// waga 
eWeightPackage2PhasePackageState[2].nID; eWeightPackage2PhasePackageState[2].nCardNumber; eWeightPackage2PhasePackageState[2].bFormPresent; eWeightPackage2PhasePackageState[2].bBottlePresent; eWeightPackage2PhasePackageState[2].bWeightOK; eWeightPackage2PhasePackageState[2].bWeighed;	eWeightPackage2PhasePackageState[2].bDosingTwoPhases; eWeightPackage2PhasePackageState[2].lrDoseVolumeSV; eWeightPackage2PhasePackageState[2].lrDoseVolumeSVSecondPhase;  eWeightPackage2PhasePackageState[2].lrDoseVolumeCV; eWeightPackage2PhasePackageState[2].lrDoseVolumeCVSecondPhase; eWeightPackage2PhasePackageState[2].nDispencerNr; eWeightPackage2PhasePackageState[2].nDispencerNrSecondPhase; eWeightPackage2PhasePackageState[2].tDispencingTime; eWeightPackage2PhasePackageState[2].tDispencingTimeSecondPhase; eWeightPackage2PhasePackageState[2].bWeighed; eWeightPackage2PhasePackageState[2].bWeightOK; eWeightPackage2PhasePackageState[2].lrWeightSV; eWeightPackage2PhasePackageState[2].lrWeightMeasuredCV; eWeightPackage2PhasePackageState[2].lrWeightCV;
eWeightPackage2PhasePackageState[1].nID; eWeightPackage2PhasePackageState[1].nCardNumber; eWeightPackage2PhasePackageState[1].bFormPresent; eWeightPackage2PhasePackageState[1].bBottlePresent; eWeightPackage2PhasePackageState[1].bWeightOK; eWeightPackage2PhasePackageState[1].bWeighed;;	eWeightPackage2PhasePackageState[1].bDosingTwoPhases; eWeightPackage2PhasePackageState[1].lrDoseVolumeSV; eWeightPackage2PhasePackageState[1].lrDoseVolumeSVSecondPhase;  eWeightPackage2PhasePackageState[1].lrDoseVolumeCV; eWeightPackage2PhasePackageState[1].lrDoseVolumeCVSecondPhase; eWeightPackage2PhasePackageState[1].nDispencerNr; eWeightPackage2PhasePackageState[1].nDispencerNrSecondPhase; eWeightPackage2PhasePackageState[1].tDispencingTime; eWeightPackage2PhasePackageState[1].tDispencingTimeSecondPhase; eWeightPackage2PhasePackageState[1].bWeighed; eWeightPackage2PhasePackageState[1].bWeightOK; eWeightPackage2PhasePackageState[1].lrWeightSV; eWeightPackage2PhasePackageState[1].lrWeightMeasuredCV; eWeightPackage2PhasePackageState[1].lrWeightCV;


/////////////////////////////////////////////////

//[1..4] Strukutra pod wagą 
eWeightPackageState[4].nID; eWeightPackageState[4].nCardNumber; eWeightPackageState[4].bFormPresent; eWeightPackageState[4].bBottlePresent; eWeightPackageState[4].bWeightOK; eWeightPackageState[4].bWeighed; 	eWeightPackageState[4].bDosingTwoPhases; eWeightPackageState[4].lrDoseVolumeSV; eWeightPackageState[4].lrDoseVolumeSVSecondPhase;  eWeightPackageState[4].lrDoseVolumeCV; eWeightPackageState[4].lrDoseVolumeCVSecondPhase; eWeightPackageState[4].nDispencerNr; eWeightPackageState[4].nDispencerNrSecondPhase; eWeightPackageState[4].tDispencingTime; eWeightPackageState[4].tDispencingTimeSecondPhase; eWeightPackageState[4].bWeighed; eWeightPackageState[4].bWeightOK; eWeightPackageState[4].lrWeightSV; eWeightPackageState[4].lrWeightMeasuredCV; eWeightPackageState[4].lrWeightCV;
eWeightPackageState[3].nID; eWeightPackageState[3].nCardNumber; eWeightPackageState[3].bFormPresent; eWeightPackageState[3].bBottlePresent; eWeightPackageState[3].bWeightOK; eWeightPackageState[3].bWeighed; 	eWeightPackageState[3].bDosingTwoPhases; eWeightPackageState[3].lrDoseVolumeSV; eWeightPackageState[3].lrDoseVolumeSVSecondPhase;  eWeightPackageState[3].lrDoseVolumeCV; eWeightPackageState[3].lrDoseVolumeCVSecondPhase; eWeightPackageState[3].nDispencerNr; eWeightPackageState[3].nDispencerNrSecondPhase; eWeightPackageState[3].tDispencingTime; eWeightPackageState[3].tDispencingTimeSecondPhase; eWeightPackageState[3].bWeighed; eWeightPackageState[3].bWeightOK; eWeightPackageState[3].lrWeightSV; eWeightPackageState[3].lrWeightMeasuredCV; eWeightPackageState[3].lrWeightCV;
eWeightPackageState[2].nID; eWeightPackageState[2].nCardNumber; eWeightPackageState[2].bFormPresent; eWeightPackageState[2].bBottlePresent; eWeightPackageState[2].bWeightOK; eWeightPackageState[2].bWeighed;	eWeightPackageState[2].bDosingTwoPhases; eWeightPackageState[2].lrDoseVolumeSV; eWeightPackageState[2].lrDoseVolumeSVSecondPhase;  eWeightPackageState[2].lrDoseVolumeCV; eWeightPackageState[2].lrDoseVolumeCVSecondPhase; eWeightPackageState[2].nDispencerNr; eWeightPackageState[2].nDispencerNrSecondPhase; eWeightPackageState[2].tDispencingTime; eWeightPackageState[2].tDispencingTimeSecondPhase; eWeightPackageState[2].bWeighed; eWeightPackageState[2].bWeightOK; eWeightPackageState[2].lrWeightSV; eWeightPackageState[2].lrWeightMeasuredCV; eWeightPackageState[2].lrWeightCV;
eWeightPackageState[1].nID; eWeightPackageState[1].nCardNumber; eWeightPackageState[1].bFormPresent; eWeightPackageState[1].bBottlePresent; eWeightPackageState[1].bWeightOK; eWeightPackageState[1].bWeighed;;	eWeightPackageState[1].bDosingTwoPhases; eWeightPackageState[1].lrDoseVolumeSV; eWeightPackageState[1].lrDoseVolumeSVSecondPhase;  eWeightPackageState[1].lrDoseVolumeCV; eWeightPackageState[1].lrDoseVolumeCVSecondPhase; eWeightPackageState[1].nDispencerNr; eWeightPackageState[1].nDispencerNrSecondPhase; eWeightPackageState[1].tDispencingTime; eWeightPackageState[1].tDispencingTimeSecondPhase; eWeightPackageState[1].bWeighed; eWeightPackageState[1].bWeightOK; eWeightPackageState[1].lrWeightSV; eWeightPackageState[1].lrWeightMeasuredCV; eWeightPackageState[1].lrWeightCV;
															
eTempState1[1].nID; eTempState1[1].nCardNumber; eTempState1[1].bFormPresent;

eBeforeLidFeeder2PackageState[4].nID;eBeforeLidFeeder2PackageState[4].nCardNumber;eBeforeLidFeeder2PackageState[4].bFormPresent;eBeforeLidFeeder2PackageState[4].bBottlePresent;eBeforeLidFeeder2PackageState[4].bLidPutted;eBeforeLidFeeder2PackageState[4].bLidPutAborted;eBeforeLidFeeder2PackageState[4].bLidPuttedOK;eBeforeLidFeeder2PackageState[4].bLidPuttedChecked;eBeforeLidFeeder2PackageState[4].bLidSealed;eBeforeLidFeeder2PackageState[4].bLidSealingAborted;
eBeforeLidFeeder2PackageState[3].nID;eBeforeLidFeeder2PackageState[3].nCardNumber;eBeforeLidFeeder2PackageState[3].bFormPresent;eBeforeLidFeeder2PackageState[3].bBottlePresent;eBeforeLidFeeder2PackageState[3].bLidPutted;eBeforeLidFeeder2PackageState[3].bLidPutAborted;eBeforeLidFeeder2PackageState[3].bLidPuttedOK;eBeforeLidFeeder2PackageState[3].bLidPuttedChecked;eBeforeLidFeeder2PackageState[3].bLidSealed;eBeforeLidFeeder2PackageState[3].bLidSealingAborted;
eBeforeLidFeeder2PackageState[2].nID;eBeforeLidFeeder2PackageState[2].nCardNumber;eBeforeLidFeeder2PackageState[2].bFormPresent;eBeforeLidFeeder2PackageState[2].bBottlePresent;eBeforeLidFeeder2PackageState[2].bLidPutted;eBeforeLidFeeder2PackageState[2].bLidPutAborted;eBeforeLidFeeder2PackageState[2].bLidPuttedOK;eBeforeLidFeeder2PackageState[2].bLidPuttedChecked;eBeforeLidFeeder2PackageState[2].bLidSealed;eBeforeLidFeeder2PackageState[2].bLidSealingAborted;
eBeforeLidFeeder2PackageState[1].nID;eBeforeLidFeeder2PackageState[1].nCardNumber;eBeforeLidFeeder2PackageState[1].bFormPresent;eBeforeLidFeeder2PackageState[1].bBottlePresent;eBeforeLidFeeder2PackageState[1].bLidPutted;eBeforeLidFeeder2PackageState[1].bLidPutAborted;eBeforeLidFeeder2PackageState[1].bLidPuttedOK;eBeforeLidFeeder2PackageState[1].bLidPuttedChecked;eBeforeLidFeeder2PackageState[1].bLidSealed;eBeforeLidFeeder2PackageState[1].bLidSealingAborted;

eBeforeLidFeederPackageState[2].nID;eBeforeLidFeederPackageState[2].nCardNumber;eBeforeLidFeederPackageState[2].bFormPresent;eBeforeLidFeederPackageState[2].bBottlePresent;eBeforeLidFeederPackageState[2].bLidPutted;eBeforeLidFeederPackageState[2].bLidPutAborted;eBeforeLidFeederPackageState[2].bLidPuttedOK;eBeforeLidFeederPackageState[2].bLidPuttedChecked;eBeforeLidFeederPackageState[2].bLidSealed;eBeforeLidFeederPackageState[2].bLidSealingAborted;
eBeforeLidFeederPackageState[1].nID;eBeforeLidFeederPackageState[1].nCardNumber;eBeforeLidFeederPackageState[1].bFormPresent;eBeforeLidFeederPackageState[1].bBottlePresent;eBeforeLidFeederPackageState[1].bLidPutted;eBeforeLidFeederPackageState[1].bLidPutAborted;eBeforeLidFeederPackageState[1].bLidPuttedOK;eBeforeLidFeederPackageState[1].bLidPuttedChecked;eBeforeLidFeederPackageState[1].bLidSealed;eBeforeLidFeederPackageState[1].bLidSealingAborted;

eLidFeederPackageState[2].nID;eLidFeederPackageState[2].nCardNumber;eLidFeederPackageState[2].bFormPresent;eLidFeederPackageState[2].bBottlePresent;eLidFeederPackageState[2].bLidPutted;eLidFeederPackageState[2].bLidPutAborted;eLidFeederPackageState[2].bLidPuttedOK;eLidFeederPackageState[2].bLidPuttedChecked;eLidFeederPackageState[2].bLidSealed;eLidFeederPackageState[2].bLidSealingAborted;
eLidFeederPackageState[1].nID;eLidFeederPackageState[1].nCardNumber;eLidFeederPackageState[1].bFormPresent;eLidFeederPackageState[1].bBottlePresent;eLidFeederPackageState[1].bLidPutted;eLidFeederPackageState[1].bLidPutAborted;eLidFeederPackageState[1].bLidPuttedOK;eLidFeederPackageState[1].bLidPuttedChecked;eLidFeederPackageState[1].bLidSealed;eLidFeederPackageState[1].bLidSealingAborted;

eAfterLidFeederPackageState[2].nID;eAfterLidFeederPackageState[2].nCardNumber;eAfterLidFeederPackageState[2].bFormPresent;eAfterLidFeederPackageState[2].bBottlePresent;eAfterLidFeederPackageState[2].bLidPutted;eAfterLidFeederPackageState[2].bLidPutAborted;eAfterLidFeederPackageState[2].bLidPuttedOK;eAfterLidFeederPackageState[2].bLidPuttedChecked;eAfterLidFeederPackageState[2].bLidSealed;eAfterLidFeederPackageState[2].bLidSealingAborted;
eAfterLidFeederPackageState[1].nID;eAfterLidFeederPackageState[1].nCardNumber;eAfterLidFeederPackageState[1].bFormPresent;eAfterLidFeederPackageState[1].bBottlePresent;eAfterLidFeederPackageState[1].bLidPutted;eAfterLidFeederPackageState[1].bLidPutAborted;eAfterLidFeederPackageState[1].bLidPuttedOK;eAfterLidFeederPackageState[1].bLidPuttedChecked;eAfterLidFeederPackageState[1].bLidSealed;eAfterLidFeederPackageState[1].bLidSealingAborted;

eBeforeLidSealerPackageState[2].nID;eBeforeLidSealerPackageState[2].nCardNumber;eBeforeLidSealerPackageState[2].bFormPresent;eBeforeLidSealerPackageState[2].bBottlePresent;eBeforeLidSealerPackageState[2].bLidPutted;eBeforeLidSealerPackageState[2].bLidPutAborted;eBeforeLidSealerPackageState[2].bLidPuttedOK;eBeforeLidSealerPackageState[2].bLidPuttedChecked;eBeforeLidSealerPackageState[2].bLidSealed;eBeforeLidSealerPackageState[2].bLidSealingAborted;
eBeforeLidSealerPackageState[1].nID;eBeforeLidSealerPackageState[1].nCardNumber;eBeforeLidSealerPackageState[1].bFormPresent;eBeforeLidSealerPackageState[1].bBottlePresent;eBeforeLidSealerPackageState[1].bLidPutted;eBeforeLidSealerPackageState[1].bLidPutAborted;eBeforeLidSealerPackageState[1].bLidPuttedOK;eBeforeLidSealerPackageState[1].bLidPuttedChecked;eBeforeLidSealerPackageState[1].bLidSealed;eBeforeLidSealerPackageState[1].bLidSealingAborted;

eLidSealerPackageState[2].nID;eLidSealerPackageState[2].nCardNumber;eLidSealerPackageState[2].bFormPresent;eLidSealerPackageState[2].bBottlePresent;eLidSealerPackageState[2].bLidPutted;eLidSealerPackageState[2].bLidPutAborted;eLidSealerPackageState[2].bLidPuttedOK;eLidSealerPackageState[2].bLidPuttedChecked;eLidSealerPackageState[2].bLidSealed;eLidSealerPackageState[2].bLidSealingAborted;
eLidSealerPackageState[1].nID;eLidSealerPackageState[1].nCardNumber;eLidSealerPackageState[1].bFormPresent;eLidSealerPackageState[1].bBottlePresent;eLidSealerPackageState[1].bLidPutted;eLidSealerPackageState[1].bLidPutAborted;eLidSealerPackageState[1].bLidPuttedOK;eLidSealerPackageState[1].bLidPuttedChecked;eLidSealerPackageState[1].bLidSealed;eLidSealerPackageState[1].bLidSealingAborted;



eBeforeGateCapSorterPackageState[1].nID;	eBeforeGateCapSorterPackageState[1].nCardNumber;	eBeforeGateCapSorterPackageState[1].bFormPresent;

eBeforeCapSorterPackageState[4].nID;	eBeforeCapSorterPackageState[4].nCardNumber;	eBeforeCapSorterPackageState[4].bFormPresent;eBeforeCapSorterPackageState[4].bBottlePresent;
eBeforeCapSorterPackageState[3].nID;	eBeforeCapSorterPackageState[3].nCardNumber;	eBeforeCapSorterPackageState[3].bFormPresent;eBeforeCapSorterPackageState[3].bBottlePresent;
eBeforeCapSorterPackageState[2].nID;	eBeforeCapSorterPackageState[2].nCardNumber;	eBeforeCapSorterPackageState[2].bFormPresent;eBeforeCapSorterPackageState[2].bBottlePresent;
eBeforeCapSorterPackageState[1].nID;	eBeforeCapSorterPackageState[1].nCardNumber;	eBeforeCapSorterPackageState[1].bFormPresent;eBeforeCapSorterPackageState[1].bBottlePresent;

eCapSorterPackageState[4].nID;	eCapSorterPackageState[4].nCardNumber;	eCapSorterPackageState[4].bFormPresent;	eCapSorterPackageState[4].bBottlePresent;
eCapSorterPackageState[3].nID;	eCapSorterPackageState[3].nCardNumber;	eCapSorterPackageState[3].bFormPresent;	eCapSorterPackageState[3].bBottlePresent;
eCapSorterPackageState[2].nID;	eCapSorterPackageState[2].nCardNumber;	eCapSorterPackageState[2].bFormPresent;	eCapSorterPackageState[2].bBottlePresent;
eCapSorterPackageState[1].nID;	eCapSorterPackageState[1].nCardNumber;	eCapSorterPackageState[1].bFormPresent;	eCapSorterPackageState[1].bBottlePresent;

eAfterCapSorterPackageState[4].nID;	eAfterCapSorterPackageState[4].nCardNumber;	eAfterCapSorterPackageState[4].bFormPresent;eAfterCapSorterPackageState[4].bBottlePresent;
eAfterCapSorterPackageState[3].nID;	eAfterCapSorterPackageState[3].nCardNumber;	eAfterCapSorterPackageState[3].bFormPresent;eAfterCapSorterPackageState[3].bBottlePresent;
eAfterCapSorterPackageState[2].nID;	eAfterCapSorterPackageState[2].nCardNumber;	eAfterCapSorterPackageState[2].bFormPresent;eAfterCapSorterPackageState[2].bBottlePresent;
eAfterCapSorterPackageState[1].nID;	eAfterCapSorterPackageState[1].nCardNumber;	eAfterCapSorterPackageState[1].bFormPresent;eAfterCapSorterPackageState[1].bBottlePresent;


eBeforeCapControlPackageState[1].nID; eBeforeCapControlPackageState[1].nCardNumber; eBeforeCapControlPackageState[1].bFormPresent;eBeforeCapControlPackageState[1].bBottlePresent;eBeforeCapControlPackageState[1].bCapPutted;	eBeforeCapControlPackageState[1].bCapOK;

// [1..12] Strukura przed zakręcarkami
eBeforeScrewers2PackageState[2].nID; eBeforeScrewers2PackageState[2].nCardNumber; eBeforeScrewers2PackageState[2].bFormPresent; eBeforeScrewers2PackageState[2].bBottlePresent;	eBeforeScrewers2PackageState[2].bCapPutted;	eBeforeScrewers2PackageState[2].bCapOK;		 eBeforeScrewers2PackageState[2].bDosingTwoPhases; eBeforeScrewers2PackageState[2].lrDoseVolumeSV; eBeforeScrewers2PackageState[2].lrDoseVolumeSVSecondPhase;  eBeforeScrewers2PackageState[2].lrDoseVolumeCV; eBeforeScrewers2PackageState[2].lrDoseVolumeCVSecondPhase; eBeforeScrewers2PackageState[2].nDispencerNr; eBeforeScrewers2PackageState[2].nDispencerNrSecondPhase; eBeforeScrewers2PackageState[2].tDispencingTime; eBeforeScrewers2PackageState[2].tDispencingTimeSecondPhase; eBeforeScrewers2PackageState[2].bWeighed; eBeforeScrewers2PackageState[2].bWeightOK; eBeforeScrewers2PackageState[2].lrWeightSV; eBeforeScrewers2PackageState[2].lrWeightMeasuredCV; eBeforeScrewers2PackageState[2].lrWeightCV; eBeforeScrewers2PackageState[2].bCapChecked;
eBeforeScrewers2PackageState[1].nID; eBeforeScrewers2PackageState[1].nCardNumber; eBeforeScrewers2PackageState[1].bFormPresent; eBeforeScrewers2PackageState[1].bBottlePresent;	eBeforeScrewers2PackageState[1].bCapPutted;	eBeforeScrewers2PackageState[1].bCapOK;		 eBeforeScrewers2PackageState[1].bDosingTwoPhases; eBeforeScrewers2PackageState[1].lrDoseVolumeSV; eBeforeScrewers2PackageState[1].lrDoseVolumeSVSecondPhase;  eBeforeScrewers2PackageState[1].lrDoseVolumeCV; eBeforeScrewers2PackageState[1].lrDoseVolumeCVSecondPhase; eBeforeScrewers2PackageState[1].nDispencerNr; eBeforeScrewers2PackageState[1].nDispencerNrSecondPhase; eBeforeScrewers2PackageState[1].tDispencingTime; eBeforeScrewers2PackageState[1].tDispencingTimeSecondPhase; eBeforeScrewers2PackageState[1].bWeighed; eBeforeScrewers2PackageState[1].bWeightOK; eBeforeScrewers2PackageState[1].lrWeightSV; eBeforeScrewers2PackageState[1].lrWeightMeasuredCV; eBeforeScrewers2PackageState[1].lrWeightCV; eBeforeScrewers2PackageState[1].bCapChecked;
eBeforeScrewersPackageState[2].nID;  eBeforeScrewersPackageState[2].nCardNumber;  eBeforeScrewersPackageState[2].bFormPresent;  eBeforeScrewersPackageState[2].bBottlePresent;	eBeforeScrewersPackageState[2].bCapPutted;	eBeforeScrewersPackageState[2].bCapOK;		 eBeforeScrewersPackageState[2].bDosingTwoPhases; eBeforeScrewersPackageState[2].lrDoseVolumeSV; eBeforeScrewersPackageState[2].lrDoseVolumeSVSecondPhase;  eBeforeScrewersPackageState[2].lrDoseVolumeCV; eBeforeScrewersPackageState[2].lrDoseVolumeCVSecondPhase; eBeforeScrewersPackageState[2].nDispencerNr; eBeforeScrewersPackageState[2].nDispencerNrSecondPhase; eBeforeScrewersPackageState[2].tDispencingTime; eBeforeScrewersPackageState[2].tDispencingTimeSecondPhase; eBeforeScrewersPackageState[2].bWeighed; eBeforeScrewersPackageState[2].bWeightOK; eBeforeScrewersPackageState[2].lrWeightSV; eBeforeScrewersPackageState[2].lrWeightMeasuredCV; eBeforeScrewersPackageState[2].lrWeightCV; eBeforeScrewersPackageState[2].bCapChecked;
eBeforeScrewersPackageState[1].nID;  eBeforeScrewersPackageState[1].nCardNumber;  eBeforeScrewersPackageState[1].bFormPresent;  eBeforeScrewersPackageState[1].bBottlePresent;	eBeforeScrewersPackageState[1].bCapPutted;	eBeforeScrewersPackageState[1].bCapOK;		 eBeforeScrewersPackageState[1].bDosingTwoPhases; eBeforeScrewersPackageState[1].lrDoseVolumeSV; eBeforeScrewersPackageState[1].lrDoseVolumeSVSecondPhase;  eBeforeScrewersPackageState[1].lrDoseVolumeCV; eBeforeScrewersPackageState[1].lrDoseVolumeCVSecondPhase; eBeforeScrewersPackageState[1].nDispencerNr; eBeforeScrewersPackageState[1].nDispencerNrSecondPhase; eBeforeScrewersPackageState[1].tDispencingTime; eBeforeScrewersPackageState[1].tDispencingTimeSecondPhase; eBeforeScrewersPackageState[1].bWeighed; eBeforeScrewersPackageState[1].bWeightOK; eBeforeScrewersPackageState[1].lrWeightSV; eBeforeScrewersPackageState[1].lrWeightMeasuredCV; eBeforeScrewersPackageState[1].lrWeightCV; eBeforeScrewersPackageState[1].bCapChecked;
				
//[1..3] Struktura pod zakręcarkami
eUnderScrewerPackageState[2].nID; eUnderScrewerPackageState[2].nCardNumber; eUnderScrewerPackageState[2].bFormPresent; eUnderScrewerPackageState[2].bBottlePresent; eUnderScrewerPackageState[2].bCapPutted; eUnderScrewerPackageState[2].bCapOK; eUnderScrewerPackageState[2].bCapGripperScrewAborted; eUnderScrewerPackageState[2].bCapGripperScrewed; eUnderScrewerPackageState[2].bDosingTwoPhases; eUnderScrewerPackageState[2].lrDoseVolumeSV; eUnderScrewerPackageState[2].lrDoseVolumeSVSecondPhase;  eUnderScrewerPackageState[2].lrDoseVolumeCV; eUnderScrewerPackageState[2].lrDoseVolumeCVSecondPhase; eUnderScrewerPackageState[2].nDispencerNr; eUnderScrewerPackageState[2].nDispencerNrSecondPhase; eUnderScrewerPackageState[2].tDispencingTime; eUnderScrewerPackageState[2].tDispencingTimeSecondPhase; eUnderScrewerPackageState[2].bWeighed; eUnderScrewerPackageState[2].bWeightOK; eUnderScrewerPackageState[12].lrWeightSV; eUnderScrewerPackageState[2].lrWeightMeasuredCV; eUnderScrewerPackageState[2].lrWeightCV; 
eUnderScrewerPackageState[1].nID; eUnderScrewerPackageState[1].nCardNumber; eUnderScrewerPackageState[1].bFormPresent; eUnderScrewerPackageState[1].bBottlePresent; eUnderScrewerPackageState[1].bCapPutted; eUnderScrewerPackageState[1].bCapOK; eUnderScrewerPackageState[1].bCapGripperScrewAborted; eUnderScrewerPackageState[1].bCapGripperScrewed; eUnderScrewerPackageState[1].bDosingTwoPhases; eUnderScrewerPackageState[1].lrDoseVolumeSV; eUnderScrewerPackageState[1].lrDoseVolumeSVSecondPhase;  eUnderScrewerPackageState[1].lrDoseVolumeCV; eUnderScrewerPackageState[1].lrDoseVolumeCVSecondPhase; eUnderScrewerPackageState[1].nDispencerNr; eUnderScrewerPackageState[1].nDispencerNrSecondPhase; eUnderScrewerPackageState[1].tDispencingTime; eUnderScrewerPackageState[1].tDispencingTimeSecondPhase; eUnderScrewerPackageState[1].bWeighed; eUnderScrewerPackageState[1].bWeightOK; eUnderScrewerPackageState[12].lrWeightSV; eUnderScrewerPackageState[1].lrWeightMeasuredCV; eUnderScrewerPackageState[1].lrWeightCV; 


// [1..12] Struktura za zakręcarkami
eAfterScrewerPackageState[2].nID; eAfterScrewerPackageState[2].nCardNumber; eAfterScrewerPackageState[2].bFormPresent; eAfterScrewerPackageState[2].bBottlePresent; eAfterScrewerPackageState[2].bCapPutted; eAfterScrewerPackageState[2].bCapOK; eAfterScrewerPackageState[2].bCapGripperScrewAborted; eAfterScrewerPackageState[2].bCapGripperScrewed; eAfterScrewerPackageState[2].bDosingTwoPhases; eAfterScrewerPackageState[2].lrDoseVolumeSV; eAfterScrewerPackageState[2].lrDoseVolumeSVSecondPhase;  eAfterScrewerPackageState[2].lrDoseVolumeCV; eAfterScrewerPackageState[2].lrDoseVolumeCVSecondPhase; eAfterScrewerPackageState[2].nDispencerNr; eAfterScrewerPackageState[2].nDispencerNrSecondPhase; eAfterScrewerPackageState[2].tDispencingTime; eAfterScrewerPackageState[2].tDispencingTimeSecondPhase; eAfterScrewerPackageState[2].bWeighed; eAfterScrewerPackageState[2].bWeightOK; eAfterScrewerPackageState[2].lrWeightSV; eAfterScrewerPackageState[2].lrWeightMeasuredCV; eAfterScrewerPackageState[2].lrWeightCV; 
eAfterScrewerPackageState[1].nID; eAfterScrewerPackageState[1].nCardNumber; eAfterScrewerPackageState[1].bFormPresent; eAfterScrewerPackageState[1].bBottlePresent; eAfterScrewerPackageState[1].bCapPutted; eAfterScrewerPackageState[1].bCapOK; eAfterScrewerPackageState[1].bCapGripperScrewAborted; eAfterScrewerPackageState[1].bCapGripperScrewed; eAfterScrewerPackageState[1].bDosingTwoPhases; eAfterScrewerPackageState[1].lrDoseVolumeSV; eAfterScrewerPackageState[1].lrDoseVolumeSVSecondPhase;  eAfterScrewerPackageState[1].lrDoseVolumeCV; eAfterScrewerPackageState[1].lrDoseVolumeCVSecondPhase; eAfterScrewerPackageState[1].nDispencerNr; eAfterScrewerPackageState[1].nDispencerNrSecondPhase; eAfterScrewerPackageState[1].tDispencingTime; eAfterScrewerPackageState[1].tDispencingTimeSecondPhase; eAfterScrewerPackageState[1].bWeighed; eAfterScrewerPackageState[1].bWeightOK; eAfterScrewerPackageState[1].lrWeightSV; eAfterScrewerPackageState[1].lrWeightMeasuredCV; eAfterScrewerPackageState[1].lrWeightCV; 

// za zakrecarmai i kontorla[1..8] 
eUnderCorrectCapPackageState[9].nID; eUnderCorrectCapPackageState[9].nCardNumber; eUnderCorrectCapPackageState[9].bFormPresent; eUnderCorrectCapPackageState[9].bBottlePresent; eUnderCorrectCapPackageState[9].bCapPutted; eUnderCorrectCapPackageState[9].bCapOK;eUnderCorrectCapPackageState[9].bCapGripperScrewAborted; eUnderCorrectCapPackageState[9].bCapGripperScrewed; eUnderCorrectCapPackageState[9].bDosingTwoPhases; eUnderCorrectCapPackageState[1].lrDoseVolumeSV; eUnderCorrectCapPackageState[1].lrDoseVolumeSVSecondPhase;  eUnderCorrectCapPackageState[1].lrDoseVolumeCV; eUnderCorrectCapPackageState[1].lrDoseVolumeCVSecondPhase; eUnderCorrectCapPackageState[8].nDispencerNr; eUnderCorrectCapPackageState[1].nDispencerNrSecondPhase; eAfterScrewerPackageState[1].tDispencingTime; eAfterScrewerPackageState[1].tDispencingTimeSecondPhase; eAfterScrewerPackageState[1].bWeighed; eAfterScrewerPackageState[1].bWeightOK; eUnderCorrectCapPackageState[1].lrWeightSV; eUnderCorrectCapPackageState[1].lrWeightMeasuredCV; eUnderCorrectCapPackageState[1].lrWeightCV; 
eUnderCorrectCapPackageState[8].nID; eUnderCorrectCapPackageState[8].nCardNumber; eUnderCorrectCapPackageState[8].bFormPresent; eUnderCorrectCapPackageState[8].bBottlePresent; eUnderCorrectCapPackageState[8].bCapPutted; eUnderCorrectCapPackageState[8].bCapOK;eUnderCorrectCapPackageState[8].bCapGripperScrewAborted; eUnderCorrectCapPackageState[8].bCapGripperScrewed; eUnderCorrectCapPackageState[8].bDosingTwoPhases; eUnderCorrectCapPackageState[1].lrDoseVolumeSV; eUnderCorrectCapPackageState[1].lrDoseVolumeSVSecondPhase;  eUnderCorrectCapPackageState[1].lrDoseVolumeCV; eUnderCorrectCapPackageState[1].lrDoseVolumeCVSecondPhase; eUnderCorrectCapPackageState[8].nDispencerNr; eUnderCorrectCapPackageState[1].nDispencerNrSecondPhase; eAfterScrewerPackageState[1].tDispencingTime; eAfterScrewerPackageState[1].tDispencingTimeSecondPhase; eAfterScrewerPackageState[1].bWeighed; eAfterScrewerPackageState[1].bWeightOK; eUnderCorrectCapPackageState[1].lrWeightSV; eUnderCorrectCapPackageState[1].lrWeightMeasuredCV; eUnderCorrectCapPackageState[1].lrWeightCV; 
eUnderCorrectCapPackageState[7].nID; eUnderCorrectCapPackageState[7].nCardNumber; eUnderCorrectCapPackageState[7].bFormPresent; eUnderCorrectCapPackageState[7].bBottlePresent; eUnderCorrectCapPackageState[7].bCapPutted; eUnderCorrectCapPackageState[7].bCapOK;eUnderCorrectCapPackageState[7].bCapGripperScrewAborted; eUnderCorrectCapPackageState[7].bCapGripperScrewed; eUnderCorrectCapPackageState[7].bDosingTwoPhases; eUnderCorrectCapPackageState[1].lrDoseVolumeSV; eUnderCorrectCapPackageState[1].lrDoseVolumeSVSecondPhase;  eUnderCorrectCapPackageState[1].lrDoseVolumeCV; eUnderCorrectCapPackageState[1].lrDoseVolumeCVSecondPhase; eUnderCorrectCapPackageState[8].nDispencerNr; eUnderCorrectCapPackageState[1].nDispencerNrSecondPhase; eAfterScrewerPackageState[1].tDispencingTime; eAfterScrewerPackageState[1].tDispencingTimeSecondPhase; eAfterScrewerPackageState[1].bWeighed; eAfterScrewerPackageState[1].bWeightOK; eUnderCorrectCapPackageState[1].lrWeightSV; eUnderCorrectCapPackageState[1].lrWeightMeasuredCV; eUnderCorrectCapPackageState[1].lrWeightCV; 
eUnderCorrectCapPackageState[6].nID; eUnderCorrectCapPackageState[6].nCardNumber; eUnderCorrectCapPackageState[6].bFormPresent; eUnderCorrectCapPackageState[6].bBottlePresent; eUnderCorrectCapPackageState[6].bCapPutted; eUnderCorrectCapPackageState[6].bCapOK;eUnderCorrectCapPackageState[6].bCapGripperScrewAborted; eUnderCorrectCapPackageState[6].bCapGripperScrewed; eUnderCorrectCapPackageState[6].bDosingTwoPhases; eUnderCorrectCapPackageState[1].lrDoseVolumeSV; eUnderCorrectCapPackageState[1].lrDoseVolumeSVSecondPhase;  eUnderCorrectCapPackageState[1].lrDoseVolumeCV; eUnderCorrectCapPackageState[1].lrDoseVolumeCVSecondPhase; eUnderCorrectCapPackageState[8].nDispencerNr; eUnderCorrectCapPackageState[1].nDispencerNrSecondPhase; eAfterScrewerPackageState[1].tDispencingTime; eAfterScrewerPackageState[1].tDispencingTimeSecondPhase; eAfterScrewerPackageState[1].bWeighed; eAfterScrewerPackageState[1].bWeightOK; eUnderCorrectCapPackageState[1].lrWeightSV; eUnderCorrectCapPackageState[1].lrWeightMeasuredCV; eUnderCorrectCapPackageState[1].lrWeightCV; 
eUnderCorrectCapPackageState[5].nID; eUnderCorrectCapPackageState[5].nCardNumber; eUnderCorrectCapPackageState[5].bFormPresent; eUnderCorrectCapPackageState[5].bBottlePresent; eUnderCorrectCapPackageState[5].bCapPutted; eUnderCorrectCapPackageState[5].bCapOK;eUnderCorrectCapPackageState[5].bCapGripperScrewAborted; eUnderCorrectCapPackageState[5].bCapGripperScrewed; eUnderCorrectCapPackageState[5].bDosingTwoPhases; eUnderCorrectCapPackageState[1].lrDoseVolumeSV; eUnderCorrectCapPackageState[1].lrDoseVolumeSVSecondPhase;  eUnderCorrectCapPackageState[1].lrDoseVolumeCV; eUnderCorrectCapPackageState[1].lrDoseVolumeCVSecondPhase; eUnderCorrectCapPackageState[8].nDispencerNr; eUnderCorrectCapPackageState[1].nDispencerNrSecondPhase; eAfterScrewerPackageState[1].tDispencingTime; eAfterScrewerPackageState[1].tDispencingTimeSecondPhase; eAfterScrewerPackageState[1].bWeighed; eAfterScrewerPackageState[1].bWeightOK; eUnderCorrectCapPackageState[1].lrWeightSV; eUnderCorrectCapPackageState[1].lrWeightMeasuredCV; eUnderCorrectCapPackageState[1].lrWeightCV; 
eUnderCorrectCapPackageState[4].nID; eUnderCorrectCapPackageState[4].nCardNumber; eUnderCorrectCapPackageState[4].bFormPresent; eUnderCorrectCapPackageState[4].bBottlePresent; eUnderCorrectCapPackageState[4].bCapPutted; eUnderCorrectCapPackageState[4].bCapOK;eUnderCorrectCapPackageState[4].bCapGripperScrewAborted; eUnderCorrectCapPackageState[4].bCapGripperScrewed; eUnderCorrectCapPackageState[4].bDosingTwoPhases; eUnderCorrectCapPackageState[1].lrDoseVolumeSV; eUnderCorrectCapPackageState[1].lrDoseVolumeSVSecondPhase;  eUnderCorrectCapPackageState[1].lrDoseVolumeCV; eUnderCorrectCapPackageState[1].lrDoseVolumeCVSecondPhase; eUnderCorrectCapPackageState[8].nDispencerNr; eUnderCorrectCapPackageState[1].nDispencerNrSecondPhase; eAfterScrewerPackageState[1].tDispencingTime; eAfterScrewerPackageState[1].tDispencingTimeSecondPhase; eAfterScrewerPackageState[1].bWeighed; eAfterScrewerPackageState[1].bWeightOK; eUnderCorrectCapPackageState[1].lrWeightSV; eUnderCorrectCapPackageState[1].lrWeightMeasuredCV; eUnderCorrectCapPackageState[1].lrWeightCV; 
eUnderCorrectCapPackageState[3].nID; eUnderCorrectCapPackageState[3].nCardNumber; eUnderCorrectCapPackageState[3].bFormPresent; eUnderCorrectCapPackageState[3].bBottlePresent; eUnderCorrectCapPackageState[3].bCapPutted; eUnderCorrectCapPackageState[3].bCapOK;eUnderCorrectCapPackageState[3].bCapGripperScrewAborted; eUnderCorrectCapPackageState[3].bCapGripperScrewed; eUnderCorrectCapPackageState[3].bDosingTwoPhases; eUnderCorrectCapPackageState[1].lrDoseVolumeSV; eUnderCorrectCapPackageState[1].lrDoseVolumeSVSecondPhase;  eUnderCorrectCapPackageState[1].lrDoseVolumeCV; eUnderCorrectCapPackageState[1].lrDoseVolumeCVSecondPhase; eUnderCorrectCapPackageState[8].nDispencerNr; eUnderCorrectCapPackageState[1].nDispencerNrSecondPhase; eAfterScrewerPackageState[1].tDispencingTime; eAfterScrewerPackageState[1].tDispencingTimeSecondPhase; eAfterScrewerPackageState[1].bWeighed; eAfterScrewerPackageState[1].bWeightOK; eUnderCorrectCapPackageState[1].lrWeightSV; eUnderCorrectCapPackageState[1].lrWeightMeasuredCV; eUnderCorrectCapPackageState[1].lrWeightCV; 
eUnderCorrectCapPackageState[2].nID; eUnderCorrectCapPackageState[2].nCardNumber; eUnderCorrectCapPackageState[2].bFormPresent; eUnderCorrectCapPackageState[2].bBottlePresent; eUnderCorrectCapPackageState[2].bCapPutted; eUnderCorrectCapPackageState[2].bCapOK;eUnderCorrectCapPackageState[2].bCapGripperScrewAborted; eUnderCorrectCapPackageState[2].bCapGripperScrewed; eUnderCorrectCapPackageState[2].bDosingTwoPhases; eUnderCorrectCapPackageState[1].lrDoseVolumeSV; eUnderCorrectCapPackageState[1].lrDoseVolumeSVSecondPhase;  eUnderCorrectCapPackageState[1].lrDoseVolumeCV; eUnderCorrectCapPackageState[1].lrDoseVolumeCVSecondPhase; eUnderCorrectCapPackageState[8].nDispencerNr; eUnderCorrectCapPackageState[1].nDispencerNrSecondPhase; eAfterScrewerPackageState[1].tDispencingTime; eAfterScrewerPackageState[1].tDispencingTimeSecondPhase; eAfterScrewerPackageState[1].bWeighed; eAfterScrewerPackageState[1].bWeightOK; eUnderCorrectCapPackageState[1].lrWeightSV; eUnderCorrectCapPackageState[1].lrWeightMeasuredCV; eUnderCorrectCapPackageState[1].lrWeightCV; 
eUnderCorrectCapPackageState[1].nID; eUnderCorrectCapPackageState[1].nCardNumber; eUnderCorrectCapPackageState[1].bFormPresent; eUnderCorrectCapPackageState[1].bBottlePresent; eUnderCorrectCapPackageState[1].bCapPutted; eUnderCorrectCapPackageState[1].bCapOK;eUnderCorrectCapPackageState[1].bCapGripperScrewAborted; eUnderCorrectCapPackageState[1].bCapGripperScrewed; eUnderCorrectCapPackageState[1].bDosingTwoPhases; eUnderCorrectCapPackageState[1].lrDoseVolumeSV; eUnderCorrectCapPackageState[1].lrDoseVolumeSVSecondPhase;  eUnderCorrectCapPackageState[1].lrDoseVolumeCV; eUnderCorrectCapPackageState[1].lrDoseVolumeCVSecondPhase; eUnderCorrectCapPackageState[8].nDispencerNr; eUnderCorrectCapPackageState[1].nDispencerNrSecondPhase; eAfterScrewerPackageState[1].tDispencingTime; eAfterScrewerPackageState[1].tDispencingTimeSecondPhase; eAfterScrewerPackageState[1].bWeighed; eAfterScrewerPackageState[1].bWeightOK; eUnderCorrectCapPackageState[1].lrWeightSV; eUnderCorrectCapPackageState[1].lrWeightMeasuredCV; eUnderCorrectCapPackageState[1].lrWeightCV; 


// [1..1] Struktura pod robotem
eRobotPackageState[2].nID; eRobotPackageState[2].nCardNumber; eRobotPackageState[2].bFormPresent; eRobotPackageState[2].bBottleTransferedToExit;  eRobotPackageState[2].bBottleTransferedToLabeler; eRobotPackageState[2].bBottlePresent; eRobotPackageState[2].bCapPutted; eRobotPackageState[2].bCapOK; eRobotPackageState[2].bCapGripperScrewAborted; eRobotPackageState[2].bCapGripperScrewed; ; eRobotPackageState[2].bDosingTwoPhases; eRobotPackageState[2].lrDoseVolumeSV; eRobotPackageState[2].lrDoseVolumeSVSecondPhase;  eRobotPackageState[2].lrDoseVolumeCV; eRobotPackageState[2].lrDoseVolumeCVSecondPhase; eRobotPackageState[2].nDispencerNr; eRobotPackageState[2].nDispencerNrSecondPhase; eRobotPackageState[2].tDispencingTime; eRobotPackageState[2].tDispencingTimeSecondPhase; eRobotPackageState[2].bWeighed; eRobotPackageState[2].bWeightOK; eRobotPackageState[2].lrWeightSV; eRobotPackageState[2].lrWeightMeasuredCV; eRobotPackageState[2].lrWeightCV;
eRobotPackageState[1].nID; eRobotPackageState[1].nCardNumber; eRobotPackageState[1].bFormPresent; eRobotPackageState[1].bBottleTransferedToExit;  eRobotPackageState[1].bBottleTransferedToLabeler; eRobotPackageState[1].bBottlePresent; eRobotPackageState[1].bCapPutted; eRobotPackageState[1].bCapOK; eRobotPackageState[1].bCapGripperScrewAborted; eRobotPackageState[1].bCapGripperScrewed; ; eRobotPackageState[1].bDosingTwoPhases; eRobotPackageState[1].lrDoseVolumeSV; eRobotPackageState[1].lrDoseVolumeSVSecondPhase;  eRobotPackageState[1].lrDoseVolumeCV; eRobotPackageState[1].lrDoseVolumeCVSecondPhase; eRobotPackageState[1].nDispencerNr; eRobotPackageState[1].nDispencerNrSecondPhase; eRobotPackageState[1].tDispencingTime; eRobotPackageState[1].tDispencingTimeSecondPhase; eRobotPackageState[1].bWeighed; eRobotPackageState[1].bWeightOK; eRobotPackageState[1].lrWeightSV; eRobotPackageState[1].lrWeightMeasuredCV; eRobotPackageState[1].lrWeightCV;
// Struktura historyczna przetransferowanych butelek
eRobotTempState[1].bFormPresent;eRobotTempState[1].bBottleTransferedToExit;eRobotTempState[1].bFormPresent;eRobotTempState[1].bBottleTransferedToLabeler;
///
eHistoryPackageState[1].bFormPresent; eHistoryPackageState[1].ncardNumber;eHistoryPackageState[1].nID; eHistoryPackageState[1].bBottlePresent; eHistoryPackageState[1].bBottleTransferedToExit; eHistoryPackageState[1].bBottleTransferedToLabeler; eHistoryPackageState[1].bCapPutted; eHistoryPackageState[1].bCapOK; eHistoryPackageState[1].bCapGripperScrewAborted; eHistoryPackageState[1].bCapGripperScrewed; eHistoryPackageState[1].bCapCorrectChecked;eHistoryPackageState[1].bCapCorrectCapOn;eHistoryPackageState[1].bCapCorrectNOK;	eHistoryPackageState[1].bDosingTwoPhases; eHistoryPackageState[1].lrDoseVolumeSV; eHistoryPackageState[1].lrDoseVolumeSVSecondPhase;  eHistoryPackageState[1].lrDoseVolumeCV; eHistoryPackageState[1].lrDoseVolumeCVSecondPhase; eHistoryPackageState[1].nDispencerNr; eHistoryPackageState[1].nDispencerNrSecondPhase; eHistoryPackageState[1].tDispencingTime; eHistoryPackageState[1].tDispencingTimeSecondPhase; eHistoryPackageState[1].bWeighed; eHistoryPackageState[1].bWeightOK; eHistoryPackageState[1].lrWeightSV; eHistoryPackageState[1].lrWeightMeasuredCV; eHistoryPackageState[1].lrWeightCV; 
eHistoryPackageState[2].bFormPresent; eHistoryPackageState[2].ncardNumber;eHistoryPackageState[2].nID; eHistoryPackageState[2].bBottlePresent; eHistoryPackageState[2].bBottleTransferedToExit; eHistoryPackageState[2].bBottleTransferedToLabeler; eHistoryPackageState[2].bCapPutted; eHistoryPackageState[2].bCapOK; eHistoryPackageState[2].bCapGripperScrewAborted; eHistoryPackageState[2].bCapGripperScrewed; eHistoryPackageState[2].bCapCorrectChecked;eHistoryPackageState[2].bCapCorrectCapOn;eHistoryPackageState[2].bCapCorrectNOK;	eHistoryPackageState[2].bDosingTwoPhases; eHistoryPackageState[2].lrDoseVolumeSV; eHistoryPackageState[2].lrDoseVolumeSVSecondPhase;  eHistoryPackageState[2].lrDoseVolumeCV; eHistoryPackageState[2].lrDoseVolumeCVSecondPhase; eHistoryPackageState[2].nDispencerNr; eHistoryPackageState[2].nDispencerNrSecondPhase; eHistoryPackageState[2].tDispencingTime; eHistoryPackageState[2].tDispencingTimeSecondPhase; eHistoryPackageState[2].bWeighed; eHistoryPackageState[2].bWeightOK; eHistoryPackageState[2].lrWeightSV; eHistoryPackageState[2].lrWeightMeasuredCV; eHistoryPackageState[2].lrWeightCV; 
eHistoryPackageState[3].bFormPresent; eHistoryPackageState[3].ncardNumber;eHistoryPackageState[3].nID; eHistoryPackageState[3].bBottlePresent; eHistoryPackageState[3].bBottleTransferedToExit; eHistoryPackageState[3].bBottleTransferedToLabeler; eHistoryPackageState[3].bCapPutted; eHistoryPackageState[3].bCapOK; eHistoryPackageState[3].bCapGripperScrewAborted; eHistoryPackageState[3].bCapGripperScrewed; eHistoryPackageState[3].bCapCorrectChecked;eHistoryPackageState[3].bCapCorrectCapOn;eHistoryPackageState[3].bCapCorrectNOK;	eHistoryPackageState[3].bDosingTwoPhases; eHistoryPackageState[3].lrDoseVolumeSV; eHistoryPackageState[3].lrDoseVolumeSVSecondPhase;  eHistoryPackageState[3].lrDoseVolumeCV; eHistoryPackageState[3].lrDoseVolumeCVSecondPhase; eHistoryPackageState[3].nDispencerNr; eHistoryPackageState[3].nDispencerNrSecondPhase; eHistoryPackageState[3].tDispencingTime; eHistoryPackageState[3].tDispencingTimeSecondPhase; eHistoryPackageState[3].bWeighed; eHistoryPackageState[3].bWeightOK; eHistoryPackageState[3].lrWeightSV; eHistoryPackageState[3].lrWeightMeasuredCV; eHistoryPackageState[3].lrWeightCV; 
eHistoryPackageState[4].bFormPresent; eHistoryPackageState[4].ncardNumber;eHistoryPackageState[4].nID; eHistoryPackageState[4].bBottlePresent; eHistoryPackageState[4].bBottleTransferedToExit; eHistoryPackageState[4].bBottleTransferedToLabeler; eHistoryPackageState[4].bCapPutted; eHistoryPackageState[4].bCapOK; eHistoryPackageState[4].bCapGripperScrewAborted; eHistoryPackageState[4].bCapGripperScrewed; eHistoryPackageState[4].bCapCorrectChecked;eHistoryPackageState[4].bCapCorrectCapOn;eHistoryPackageState[4].bCapCorrectNOK;	eHistoryPackageState[4].bDosingTwoPhases; eHistoryPackageState[4].lrDoseVolumeSV; eHistoryPackageState[4].lrDoseVolumeSVSecondPhase;  eHistoryPackageState[4].lrDoseVolumeCV; eHistoryPackageState[4].lrDoseVolumeCVSecondPhase; eHistoryPackageState[4].nDispencerNr; eHistoryPackageState[4].nDispencerNrSecondPhase; eHistoryPackageState[4].tDispencingTime; eHistoryPackageState[4].tDispencingTimeSecondPhase; eHistoryPackageState[4].bWeighed; eHistoryPackageState[4].bWeightOK; eHistoryPackageState[4].lrWeightSV; eHistoryPackageState[4].lrWeightMeasuredCV; eHistoryPackageState[4].lrWeightCV; 
eHistoryPackageState[5].bFormPresent; eHistoryPackageState[5].ncardNumber;eHistoryPackageState[5].nID; eHistoryPackageState[5].bBottlePresent; eHistoryPackageState[5].bBottleTransferedToExit; eHistoryPackageState[5].bBottleTransferedToLabeler; eHistoryPackageState[5].bCapPutted; eHistoryPackageState[5].bCapOK; eHistoryPackageState[5].bCapGripperScrewAborted; eHistoryPackageState[5].bCapGripperScrewed; eHistoryPackageState[5].bCapCorrectChecked;eHistoryPackageState[5].bCapCorrectCapOn;eHistoryPackageState[5].bCapCorrectNOK;	eHistoryPackageState[5].bDosingTwoPhases; eHistoryPackageState[5].lrDoseVolumeSV; eHistoryPackageState[5].lrDoseVolumeSVSecondPhase;  eHistoryPackageState[5].lrDoseVolumeCV; eHistoryPackageState[5].lrDoseVolumeCVSecondPhase; eHistoryPackageState[5].nDispencerNr; eHistoryPackageState[5].nDispencerNrSecondPhase; eHistoryPackageState[5].tDispencingTime; eHistoryPackageState[5].tDispencingTimeSecondPhase; eHistoryPackageState[5].bWeighed; eHistoryPackageState[5].bWeightOK; eHistoryPackageState[5].lrWeightSV; eHistoryPackageState[5].lrWeightMeasuredCV; eHistoryPackageState[5].lrWeightCV; 
eHistoryPackageState[6].bFormPresent; eHistoryPackageState[6].ncardNumber;eHistoryPackageState[6].nID; eHistoryPackageState[6].bBottlePresent; eHistoryPackageState[6].bBottleTransferedToExit; eHistoryPackageState[6].bBottleTransferedToLabeler; eHistoryPackageState[6].bCapPutted; eHistoryPackageState[6].bCapOK; eHistoryPackageState[6].bCapGripperScrewAborted; eHistoryPackageState[6].bCapGripperScrewed; eHistoryPackageState[6].bCapCorrectChecked;eHistoryPackageState[6].bCapCorrectCapOn;eHistoryPackageState[6].bCapCorrectNOK;	eHistoryPackageState[6].bDosingTwoPhases; eHistoryPackageState[6].lrDoseVolumeSV; eHistoryPackageState[6].lrDoseVolumeSVSecondPhase;  eHistoryPackageState[6].lrDoseVolumeCV; eHistoryPackageState[6].lrDoseVolumeCVSecondPhase; eHistoryPackageState[6].nDispencerNr; eHistoryPackageState[6].nDispencerNrSecondPhase; eHistoryPackageState[6].tDispencingTime; eHistoryPackageState[6].tDispencingTimeSecondPhase; eHistoryPackageState[6].bWeighed; eHistoryPackageState[6].bWeightOK; eHistoryPackageState[6].lrWeightSV; eHistoryPackageState[6].lrWeightMeasuredCV; eHistoryPackageState[6].lrWeightCV; 



(*****************KONIEC ZAPISYWANIE RFID*********************)
//Kasowanie tablicy RFID
IF  bRFIDArrayClear (*OR bCycleReseting*) THEN 
			FOR i := 1 TO 100 DO
	 					eRFID[i] := eClearPackageState;
			END_FOR	
			bRFIDArrayClear := FALSE;
END_IF


IF bDeletebBottleTransferedToExit THEN // Do testów
	FOR i:=1 TO 100 DO
		eRFID[i].bBottleTransferedToExit:=FALSE;
	END_FOR
	bDeletebBottleTransferedToExit := FALSE;
END_IF
																																																																																																																																																																																																																																																											nCheckWeiginhForm ;
eRFID[1].nCardNumber; eRFID[1].bCapCorrectChecked;	eRFID[1].bCapCorrectCheckCameraOK;		eRFID[1].bCapCorrectCheckCameraChecked;			eRFID[1].bCapCorrectCapOn; eRFID[1].bCapCorrectNOK;  eRFID[1].bFormPresent; eRFID[1].bBottlePresent; eRFID[1].bDosingTwoPhases; eRFID[1].nDispencerNr; eRFID[1].nDispencerNrSecondPhase; eRFID[1].lrDoseVolumeSV; eRFID[1].lrDoseVolumeCV; eRFID[1].lrDoseVolumeSVSecondPhase; eRFID[1].lrDoseVolumeCVSecondPhase;			eRFID[1].bDosed; 	eRFID[1].bDoseAborted; eRFID[1].bWeighed; eRFID[1].lrWeightSV; eRFID[1].lrWeightCV; eRFID[1].lrWeightMeasuredCV; eRFID[1].bWeightOK; eRFID[1].bCapPutted; eRFID[1].bCapChecked; eRFID[1].bCapOK; eRFID[1].bCapGripperScrewed; eRFID[1].bCapGripperScrewAborted; eRFID[1].bBottleTransferedToExit; eRFID[1].bBottleTransferedToLabeler;  eRFID[1].lrWeightDif; eRFID[1].lrMinWeightCV; eRFID[1].lrMaxWeightCV;
eRFID[2].nCardNumber; eRFID[2].bCapCorrectChecked;	eRFID[2].bCapCorrectCheckCameraOK;		eRFID[2].bCapCorrectCheckCameraChecked;			eRFID[2].bCapCorrectCapOn; eRFID[2].bCapCorrectNOK;  eRFID[2].bFormPresent; eRFID[2].bBottlePresent; eRFID[2].bDosingTwoPhases; eRFID[2].nDispencerNr; eRFID[2].nDispencerNrSecondPhase; eRFID[2].lrDoseVolumeSV; eRFID[2].lrDoseVolumeCV; eRFID[2].lrDoseVolumeSVSecondPhase; eRFID[2].lrDoseVolumeCVSecondPhase;			eRFID[2].bDosed; 	eRFID[2].bDoseAborted; eRFID[2].bWeighed; eRFID[2].lrWeightSV; eRFID[2].lrWeightCV; eRFID[2].lrWeightMeasuredCV; eRFID[2].bWeightOK; eRFID[2].bCapPutted; eRFID[2].bCapChecked; eRFID[2].bCapOK; eRFID[2].bCapGripperScrewed; eRFID[2].bCapGripperScrewAborted; eRFID[2].bBottleTransferedToExit; eRFID[2].bBottleTransferedToLabeler;  eRFID[2].lrWeightDif; eRFID[2].lrMinWeightCV; eRFID[2].lrMaxWeightCV;
eRFID[3].nCardNumber; eRFID[3].bCapCorrectChecked;	eRFID[3].bCapCorrectCheckCameraOK;		eRFID[3].bCapCorrectCheckCameraChecked;			eRFID[3].bCapCorrectCapOn; eRFID[3].bCapCorrectNOK;  eRFID[3].bFormPresent; eRFID[3].bBottlePresent; eRFID[3].bDosingTwoPhases; eRFID[3].nDispencerNr; eRFID[3].nDispencerNrSecondPhase; eRFID[3].lrDoseVolumeSV; eRFID[3].lrDoseVolumeCV; eRFID[3].lrDoseVolumeSVSecondPhase; eRFID[3].lrDoseVolumeCVSecondPhase;			eRFID[3].bDosed; 	eRFID[3].bDoseAborted; eRFID[3].bWeighed; eRFID[3].lrWeightSV; eRFID[3].lrWeightCV; eRFID[3].lrWeightMeasuredCV; eRFID[3].bWeightOK; eRFID[3].bCapPutted; eRFID[3].bCapChecked; eRFID[3].bCapOK; eRFID[3].bCapGripperScrewed; eRFID[3].bCapGripperScrewAborted; eRFID[3].bBottleTransferedToExit; eRFID[3].bBottleTransferedToLabeler;  eRFID[3].lrWeightDif; eRFID[3].lrMinWeightCV; eRFID[3].lrMaxWeightCV;
eRFID[4].nCardNumber; eRFID[4].bCapCorrectChecked;	eRFID[4].bCapCorrectCheckCameraOK;		eRFID[4].bCapCorrectCheckCameraChecked;			eRFID[4].bCapCorrectCapOn; eRFID[4].bCapCorrectNOK;  eRFID[4].bFormPresent; eRFID[4].bBottlePresent; eRFID[4].bDosingTwoPhases; eRFID[4].nDispencerNr; eRFID[4].nDispencerNrSecondPhase; eRFID[4].lrDoseVolumeSV; eRFID[4].lrDoseVolumeCV; eRFID[4].lrDoseVolumeSVSecondPhase; eRFID[4].lrDoseVolumeCVSecondPhase;			eRFID[4].bDosed; 	eRFID[4].bDoseAborted; eRFID[4].bWeighed; eRFID[4].lrWeightSV; eRFID[4].lrWeightCV; eRFID[4].lrWeightMeasuredCV; eRFID[4].bWeightOK; eRFID[4].bCapPutted; eRFID[4].bCapChecked; eRFID[4].bCapOK; eRFID[4].bCapGripperScrewed; eRFID[4].bCapGripperScrewAborted; eRFID[4].bBottleTransferedToExit; eRFID[4].bBottleTransferedToLabeler;  eRFID[4].lrWeightDif; eRFID[4].lrMinWeightCV; eRFID[4].lrMaxWeightCV;
eRFID[5].nCardNumber; eRFID[5].bCapCorrectChecked;	eRFID[5].bCapCorrectCheckCameraOK;		eRFID[5].bCapCorrectCheckCameraChecked;			eRFID[5].bCapCorrectCapOn; eRFID[5].bCapCorrectNOK;  eRFID[5].bFormPresent; eRFID[5].bBottlePresent; eRFID[5].bDosingTwoPhases; eRFID[5].nDispencerNr; eRFID[5].nDispencerNrSecondPhase; eRFID[5].lrDoseVolumeSV; eRFID[5].lrDoseVolumeCV; eRFID[5].lrDoseVolumeSVSecondPhase; eRFID[5].lrDoseVolumeCVSecondPhase;			eRFID[5].bDosed; 	eRFID[5].bDoseAborted; eRFID[5].bWeighed; eRFID[5].lrWeightSV; eRFID[5].lrWeightCV; eRFID[5].lrWeightMeasuredCV; eRFID[5].bWeightOK; eRFID[5].bCapPutted; eRFID[5].bCapChecked; eRFID[5].bCapOK; eRFID[5].bCapGripperScrewed; eRFID[5].bCapGripperScrewAborted; eRFID[5].bBottleTransferedToExit; eRFID[5].bBottleTransferedToLabeler;  eRFID[5].lrWeightDif; eRFID[5].lrMinWeightCV; eRFID[5].lrMaxWeightCV;
eRFID[6].nCardNumber; eRFID[6].bCapCorrectChecked;	eRFID[6].bCapCorrectCheckCameraOK;		eRFID[6].bCapCorrectCheckCameraChecked;			eRFID[6].bCapCorrectCapOn; eRFID[6].bCapCorrectNOK;  eRFID[6].bFormPresent; eRFID[6].bBottlePresent; eRFID[6].bDosingTwoPhases; eRFID[6].nDispencerNr; eRFID[6].nDispencerNrSecondPhase; eRFID[6].lrDoseVolumeSV; eRFID[6].lrDoseVolumeCV; eRFID[6].lrDoseVolumeSVSecondPhase; eRFID[6].lrDoseVolumeCVSecondPhase;			eRFID[6].bDosed; 	eRFID[6].bDoseAborted; eRFID[6].bWeighed; eRFID[6].lrWeightSV; eRFID[6].lrWeightCV; eRFID[6].lrWeightMeasuredCV; eRFID[6].bWeightOK; eRFID[6].bCapPutted; eRFID[6].bCapChecked; eRFID[6].bCapOK; eRFID[6].bCapGripperScrewed; eRFID[6].bCapGripperScrewAborted; eRFID[6].bBottleTransferedToExit; eRFID[6].bBottleTransferedToLabeler;  eRFID[6].lrWeightDif; eRFID[6].lrMinWeightCV; eRFID[6].lrMaxWeightCV;
eRFID[7].nCardNumber; eRFID[7].bCapCorrectChecked;	eRFID[7].bCapCorrectCheckCameraOK;		eRFID[7].bCapCorrectCheckCameraChecked;			eRFID[7].bCapCorrectCapOn; eRFID[7].bCapCorrectNOK;  eRFID[7].bFormPresent; eRFID[7].bBottlePresent; eRFID[7].bDosingTwoPhases; eRFID[7].nDispencerNr; eRFID[7].nDispencerNrSecondPhase; eRFID[7].lrDoseVolumeSV; eRFID[7].lrDoseVolumeCV; eRFID[7].lrDoseVolumeSVSecondPhase; eRFID[7].lrDoseVolumeCVSecondPhase;			eRFID[7].bDosed; 	eRFID[7].bDoseAborted; eRFID[7].bWeighed; eRFID[7].lrWeightSV; eRFID[7].lrWeightCV; eRFID[7].lrWeightMeasuredCV; eRFID[7].bWeightOK; eRFID[7].bCapPutted; eRFID[7].bCapChecked; eRFID[7].bCapOK; eRFID[7].bCapGripperScrewed; eRFID[7].bCapGripperScrewAborted; eRFID[7].bBottleTransferedToExit; eRFID[7].bBottleTransferedToLabeler;  eRFID[7].lrWeightDif; eRFID[7].lrMinWeightCV; eRFID[7].lrMaxWeightCV;
eRFID[8].nCardNumber; eRFID[8].bCapCorrectChecked;	eRFID[8].bCapCorrectCheckCameraOK;		eRFID[8].bCapCorrectCheckCameraChecked;			eRFID[8].bCapCorrectCapOn; eRFID[8].bCapCorrectNOK;  eRFID[8].bFormPresent; eRFID[8].bBottlePresent; eRFID[8].bDosingTwoPhases; eRFID[8].nDispencerNr; eRFID[8].nDispencerNrSecondPhase; eRFID[8].lrDoseVolumeSV; eRFID[8].lrDoseVolumeCV; eRFID[8].lrDoseVolumeSVSecondPhase; eRFID[8].lrDoseVolumeCVSecondPhase; 			eRFID[8].bDosed; 	eRFID[8].bDoseAborted; eRFID[8].bWeighed; eRFID[8].lrWeightSV; eRFID[8].lrWeightCV; eRFID[8].lrWeightMeasuredCV; eRFID[8].bWeightOK; eRFID[8].bCapPutted; eRFID[8].bCapChecked; eRFID[8].bCapOK; eRFID[8].bCapGripperScrewed; eRFID[8].bCapGripperScrewAborted; eRFID[8].bBottleTransferedToExit; eRFID[8].bBottleTransferedToLabeler;  eRFID[8].lrWeightDif; eRFID[8].lrMinWeightCV; eRFID[8].lrMaxWeightCV;
eRFID[9].nCardNumber; eRFID[9].bCapCorrectChecked;	eRFID[9].bCapCorrectCheckCameraOK;		eRFID[9].bCapCorrectCheckCameraChecked;			eRFID[9].bCapCorrectCapOn; eRFID[9].bCapCorrectNOK;  eRFID[9].bFormPresent; eRFID[9].bBottlePresent; eRFID[9].bDosingTwoPhases; eRFID[9].nDispencerNr; eRFID[9].nDispencerNrSecondPhase; eRFID[9].lrDoseVolumeSV; eRFID[9].lrDoseVolumeCV; eRFID[9].lrDoseVolumeSVSecondPhase; eRFID[9].lrDoseVolumeCVSecondPhase; 			eRFID[9].bDosed; 	eRFID[9].bDoseAborted; eRFID[9].bWeighed; eRFID[9].lrWeightSV; eRFID[9].lrWeightCV; eRFID[9].lrWeightMeasuredCV; eRFID[9].bWeightOK; eRFID[9].bCapPutted; eRFID[9].bCapChecked; eRFID[9].bCapOK; eRFID[9].bCapGripperScrewed; eRFID[9].bCapGripperScrewAborted; eRFID[9].bBottleTransferedToExit; eRFID[9].bBottleTransferedToLabeler;  eRFID[9].lrWeightDif; eRFID[9].lrMinWeightCV; eRFID[9].lrMaxWeightCV;
eRFID[10].nCardNumber;eRFID[10].bCapCorrectChecked;	eRFID[10].bCapCorrectCheckCameraOK;		eRFID[10].bCapCorrectCheckCameraChecked;		eRFID[10].bCapCorrectCapOn;eRFID[10].bCapCorrectNOK; eRFID[10].bFormPresent; eRFID[10].bBottlePresent; eRFID[10].bDosingTwoPhases; eRFID[10].nDispencerNr; eRFID[10].nDispencerNrSecondPhase; eRFID[10].lrDoseVolumeSV; eRFID[10].lrDoseVolumeCV; eRFID[10].lrDoseVolumeSVSecondPhase; eRFID[10].lrDoseVolumeCVSecondPhase; eRFID[10].bDosed;	eRFID[10].bDoseAborted; eRFID[10].bWeighed; eRFID[10].lrWeightSV; eRFID[10].lrWeightCV; eRFID[10].lrWeightMeasuredCV; eRFID[10].bWeightOK; eRFID[10].bCapPutted; eRFID[10].bCapChecked; eRFID[10].bCapOK; eRFID[10].bCapGripperScrewed; eRFID[10].bCapGripperScrewAborted; eRFID[10].bBottleTransferedToExit; eRFID[10].bBottleTransferedToLabeler; eRFID[10].lrWeightDif; eRFID[10].lrMinWeightCV;eRFID[10].lrMaxWeightCV;
eRFID[11].nCardNumber;eRFID[11].bCapCorrectChecked;	eRFID[11].bCapCorrectCheckCameraOK;		eRFID[11].bCapCorrectCheckCameraChecked;		eRFID[11].bCapCorrectCapOn;eRFID[11].bCapCorrectNOK; eRFID[11].bFormPresent; eRFID[11].bBottlePresent; eRFID[11].bDosingTwoPhases; eRFID[11].nDispencerNr; eRFID[11].nDispencerNrSecondPhase; eRFID[11].lrDoseVolumeSV; eRFID[11].lrDoseVolumeCV; eRFID[11].lrDoseVolumeSVSecondPhase; eRFID[11].lrDoseVolumeCVSecondPhase; eRFID[11].bDosed;	eRFID[11].bDoseAborted; eRFID[11].bWeighed; eRFID[11].lrWeightSV; eRFID[11].lrWeightCV; eRFID[11].lrWeightMeasuredCV; eRFID[11].bWeightOK; eRFID[11].bCapPutted; eRFID[11].bCapChecked; eRFID[11].bCapOK; eRFID[11].bCapGripperScrewed; eRFID[11].bCapGripperScrewAborted; eRFID[11].bBottleTransferedToExit; eRFID[11].bBottleTransferedToLabeler; eRFID[11].lrWeightDif; eRFID[11].lrMinWeightCV;eRFID[11].lrMaxWeightCV;
eRFID[12].nCardNumber;eRFID[12].bCapCorrectChecked;	eRFID[12].bCapCorrectCheckCameraOK;		eRFID[12].bCapCorrectCheckCameraChecked;		eRFID[12].bCapCorrectCapOn;eRFID[12].bCapCorrectNOK; eRFID[12].bFormPresent; eRFID[12].bBottlePresent; eRFID[12].bDosingTwoPhases; eRFID[12].nDispencerNr; eRFID[12].nDispencerNrSecondPhase; eRFID[12].lrDoseVolumeSV; eRFID[12].lrDoseVolumeCV; eRFID[12].lrDoseVolumeSVSecondPhase; eRFID[12].lrDoseVolumeCVSecondPhase; eRFID[12].bDosed;	eRFID[12].bDoseAborted; eRFID[12].bWeighed; eRFID[12].lrWeightSV; eRFID[12].lrWeightCV; eRFID[12].lrWeightMeasuredCV; eRFID[12].bWeightOK; eRFID[12].bCapPutted; eRFID[12].bCapChecked; eRFID[12].bCapOK; eRFID[12].bCapGripperScrewed; eRFID[12].bCapGripperScrewAborted; eRFID[12].bBottleTransferedToExit; eRFID[12].bBottleTransferedToLabeler; eRFID[12].lrWeightDif; eRFID[12].lrMinWeightCV;eRFID[12].lrMaxWeightCV;
eRFID[13].nCardNumber;eRFID[13].bCapCorrectChecked;	eRFID[13].bCapCorrectCheckCameraOK;		eRFID[13].bCapCorrectCheckCameraChecked;		eRFID[13].bCapCorrectCapOn;eRFID[13].bCapCorrectNOK; eRFID[13].bFormPresent; eRFID[13].bBottlePresent; eRFID[13].bDosingTwoPhases; eRFID[13].nDispencerNr; eRFID[13].nDispencerNrSecondPhase; eRFID[13].lrDoseVolumeSV; eRFID[13].lrDoseVolumeCV; eRFID[13].lrDoseVolumeSVSecondPhase; eRFID[13].lrDoseVolumeCVSecondPhase; eRFID[13].bDosed;	eRFID[13].bDoseAborted; eRFID[13].bWeighed; eRFID[13].lrWeightSV; eRFID[13].lrWeightCV; eRFID[13].lrWeightMeasuredCV; eRFID[13].bWeightOK; eRFID[13].bCapPutted; eRFID[13].bCapChecked; eRFID[13].bCapOK; eRFID[13].bCapGripperScrewed; eRFID[13].bCapGripperScrewAborted; eRFID[13].bBottleTransferedToExit; eRFID[13].bBottleTransferedToLabeler; eRFID[13].lrWeightDif; eRFID[13].lrMinWeightCV;eRFID[13].lrMaxWeightCV;
eRFID[14].nCardNumber;eRFID[14].bCapCorrectChecked;	eRFID[14].bCapCorrectCheckCameraOK;		eRFID[14].bCapCorrectCheckCameraChecked;		eRFID[14].bCapCorrectCapOn;eRFID[14].bCapCorrectNOK; eRFID[14].bFormPresent; eRFID[14].bBottlePresent; eRFID[14].bDosingTwoPhases; eRFID[14].nDispencerNr; eRFID[14].nDispencerNrSecondPhase; eRFID[14].lrDoseVolumeSV; eRFID[14].lrDoseVolumeCV; eRFID[14].lrDoseVolumeSVSecondPhase; eRFID[14].lrDoseVolumeCVSecondPhase; eRFID[14].bDosed;	eRFID[14].bDoseAborted; eRFID[14].bWeighed; eRFID[14].lrWeightSV; eRFID[14].lrWeightCV; eRFID[14].lrWeightMeasuredCV; eRFID[14].bWeightOK; eRFID[14].bCapPutted; eRFID[14].bCapChecked; eRFID[14].bCapOK; eRFID[14].bCapGripperScrewed; eRFID[14].bCapGripperScrewAborted; eRFID[14].bBottleTransferedToExit; eRFID[14].bBottleTransferedToLabeler; eRFID[14].lrWeightDif; eRFID[14].lrMinWeightCV;eRFID[14].lrMaxWeightCV;
eRFID[15].nCardNumber;eRFID[15].bCapCorrectChecked;	eRFID[15].bCapCorrectCheckCameraOK;		eRFID[15].bCapCorrectCheckCameraChecked;		eRFID[15].bCapCorrectCapOn;eRFID[15].bCapCorrectNOK; eRFID[15].bFormPresent; eRFID[15].bBottlePresent; eRFID[15].bDosingTwoPhases; eRFID[15].nDispencerNr; eRFID[15].nDispencerNrSecondPhase; eRFID[15].lrDoseVolumeSV; eRFID[15].lrDoseVolumeCV; eRFID[15].lrDoseVolumeSVSecondPhase; eRFID[15].lrDoseVolumeCVSecondPhase; eRFID[15].bDosed;	eRFID[15].bDoseAborted; eRFID[15].bWeighed; eRFID[15].lrWeightSV; eRFID[15].lrWeightCV; eRFID[15].lrWeightMeasuredCV; eRFID[15].bWeightOK; eRFID[15].bCapPutted; eRFID[15].bCapChecked; eRFID[15].bCapOK; eRFID[15].bCapGripperScrewed; eRFID[15].bCapGripperScrewAborted; eRFID[15].bBottleTransferedToExit; eRFID[15].bBottleTransferedToLabeler; eRFID[15].lrWeightDif; eRFID[15].lrMinWeightCV;eRFID[15].lrMaxWeightCV;
eRFID[16].nCardNumber;eRFID[16].bCapCorrectChecked;	eRFID[16].bCapCorrectCheckCameraOK;		eRFID[16].bCapCorrectCheckCameraChecked;		eRFID[16].bCapCorrectCapOn;eRFID[16].bCapCorrectNOK; eRFID[16].bFormPresent; eRFID[16].bBottlePresent; eRFID[16].bDosingTwoPhases; eRFID[16].nDispencerNr; eRFID[16].nDispencerNrSecondPhase; eRFID[16].lrDoseVolumeSV; eRFID[16].lrDoseVolumeCV; eRFID[16].lrDoseVolumeSVSecondPhase; eRFID[16].lrDoseVolumeCVSecondPhase; eRFID[16].bDosed;	eRFID[16].bDoseAborted; eRFID[16].bWeighed; eRFID[16].lrWeightSV; eRFID[16].lrWeightCV; eRFID[16].lrWeightMeasuredCV; eRFID[16].bWeightOK; eRFID[16].bCapPutted; eRFID[16].bCapChecked; eRFID[16].bCapOK; eRFID[16].bCapGripperScrewed; eRFID[16].bCapGripperScrewAborted; eRFID[16].bBottleTransferedToExit; eRFID[16].bBottleTransferedToLabeler; eRFID[16].lrWeightDif; eRFID[16].lrMinWeightCV;eRFID[16].lrMaxWeightCV;
eRFID[17].nCardNumber;eRFID[17].bCapCorrectChecked;	eRFID[17].bCapCorrectCheckCameraOK;		eRFID[17].bCapCorrectCheckCameraChecked;		eRFID[17].bCapCorrectCapOn;eRFID[17].bCapCorrectNOK; eRFID[17].bFormPresent; eRFID[17].bBottlePresent; eRFID[17].bDosingTwoPhases; eRFID[17].nDispencerNr; eRFID[17].nDispencerNrSecondPhase; eRFID[17].lrDoseVolumeSV; eRFID[17].lrDoseVolumeCV; eRFID[17].lrDoseVolumeSVSecondPhase; eRFID[17].lrDoseVolumeCVSecondPhase; eRFID[17].bDosed;	eRFID[17].bDoseAborted; eRFID[17].bWeighed; eRFID[17].lrWeightSV; eRFID[17].lrWeightCV; eRFID[17].lrWeightMeasuredCV; eRFID[17].bWeightOK; eRFID[17].bCapPutted; eRFID[17].bCapChecked; eRFID[17].bCapOK; eRFID[17].bCapGripperScrewed; eRFID[17].bCapGripperScrewAborted; eRFID[17].bBottleTransferedToExit; eRFID[17].bBottleTransferedToLabeler; eRFID[17].lrWeightDif; eRFID[17].lrMinWeightCV;eRFID[17].lrMaxWeightCV;
eRFID[18].nCardNumber;eRFID[18].bCapCorrectChecked;	eRFID[18].bCapCorrectCheckCameraOK;		eRFID[18].bCapCorrectCheckCameraChecked;		eRFID[18].bCapCorrectCapOn;eRFID[18].bCapCorrectNOK; eRFID[18].bFormPresent; eRFID[18].bBottlePresent; eRFID[18].bDosingTwoPhases; eRFID[18].nDispencerNr; eRFID[18].nDispencerNrSecondPhase; eRFID[18].lrDoseVolumeSV; eRFID[18].lrDoseVolumeCV; eRFID[18].lrDoseVolumeSVSecondPhase; eRFID[18].lrDoseVolumeCVSecondPhase; eRFID[18].bDosed;	eRFID[18].bDoseAborted; eRFID[18].bWeighed; eRFID[18].lrWeightSV; eRFID[18].lrWeightCV; eRFID[18].lrWeightMeasuredCV; eRFID[18].bWeightOK; eRFID[18].bCapPutted; eRFID[18].bCapChecked; eRFID[18].bCapOK; eRFID[18].bCapGripperScrewed; eRFID[18].bCapGripperScrewAborted; eRFID[18].bBottleTransferedToExit; eRFID[18].bBottleTransferedToLabeler; eRFID[18].lrWeightDif; eRFID[18].lrMinWeightCV;eRFID[18].lrMaxWeightCV;
eRFID[19].nCardNumber;eRFID[19].bCapCorrectChecked;	eRFID[19].bCapCorrectCheckCameraOK;		eRFID[19].bCapCorrectCheckCameraChecked;		eRFID[19].bCapCorrectCapOn;eRFID[19].bCapCorrectNOK; eRFID[19].bFormPresent; eRFID[19].bBottlePresent; eRFID[19].bDosingTwoPhases; eRFID[19].nDispencerNr; eRFID[19].nDispencerNrSecondPhase; eRFID[19].lrDoseVolumeSV; eRFID[19].lrDoseVolumeCV; eRFID[19].lrDoseVolumeSVSecondPhase; eRFID[19].lrDoseVolumeCVSecondPhase; eRFID[19].bDosed;	eRFID[19].bDoseAborted; eRFID[19].bWeighed; eRFID[19].lrWeightSV; eRFID[19].lrWeightCV; eRFID[19].lrWeightMeasuredCV; eRFID[19].bWeightOK; eRFID[19].bCapPutted; eRFID[19].bCapChecked; eRFID[19].bCapOK; eRFID[19].bCapGripperScrewed; eRFID[19].bCapGripperScrewAborted; eRFID[19].bBottleTransferedToExit; eRFID[19].bBottleTransferedToLabeler; eRFID[19].lrWeightDif; eRFID[19].lrMinWeightCV;eRFID[19].lrMaxWeightCV;
eRFID[20].nCardNumber;eRFID[20].bCapCorrectChecked;	eRFID[20].bCapCorrectCheckCameraOK;		eRFID[20].bCapCorrectCheckCameraChecked;		eRFID[20].bCapCorrectCapOn;eRFID[20].bCapCorrectNOK; eRFID[20].bFormPresent; eRFID[20].bBottlePresent; eRFID[20].bDosingTwoPhases; eRFID[20].nDispencerNr; eRFID[20].nDispencerNrSecondPhase; eRFID[20].lrDoseVolumeSV; eRFID[20].lrDoseVolumeCV; eRFID[20].lrDoseVolumeSVSecondPhase; eRFID[20].lrDoseVolumeCVSecondPhase; eRFID[20].bDosed;	eRFID[20].bDoseAborted; eRFID[20].bWeighed; eRFID[20].lrWeightSV; eRFID[20].lrWeightCV; eRFID[20].lrWeightMeasuredCV; eRFID[20].bWeightOK; eRFID[20].bCapPutted; eRFID[20].bCapChecked; eRFID[20].bCapOK; eRFID[20].bCapGripperScrewed; eRFID[20].bCapGripperScrewAborted; eRFID[20].bBottleTransferedToExit; eRFID[20].bBottleTransferedToLabeler; eRFID[20].lrWeightDif; eRFID[20].lrMinWeightCV;eRFID[20].lrMaxWeightCV;
eRFID[21].nCardNumber;eRFID[21].bCapCorrectChecked;	eRFID[21].bCapCorrectCheckCameraOK;		eRFID[21].bCapCorrectCheckCameraChecked;		eRFID[21].bCapCorrectCapOn;eRFID[21].bCapCorrectNOK; eRFID[21].bFormPresent; eRFID[21].bBottlePresent; eRFID[21].bDosingTwoPhases; eRFID[21].nDispencerNr; eRFID[21].nDispencerNrSecondPhase; eRFID[21].lrDoseVolumeSV; eRFID[21].lrDoseVolumeCV; eRFID[21].lrDoseVolumeSVSecondPhase; eRFID[21].lrDoseVolumeCVSecondPhase; eRFID[21].bDosed;	eRFID[21].bDoseAborted; eRFID[21].bWeighed; eRFID[21].lrWeightSV; eRFID[21].lrWeightCV; eRFID[21].lrWeightMeasuredCV; eRFID[21].bWeightOK; eRFID[21].bCapPutted; eRFID[21].bCapChecked; eRFID[21].bCapOK; eRFID[21].bCapGripperScrewed; eRFID[21].bCapGripperScrewAborted; eRFID[21].bBottleTransferedToExit; eRFID[21].bBottleTransferedToLabeler; eRFID[21].lrWeightDif; eRFID[21].lrMinWeightCV;eRFID[21].lrMaxWeightCV;
eRFID[22].nCardNumber;eRFID[22].bCapCorrectChecked;	eRFID[22].bCapCorrectCheckCameraOK;		eRFID[22].bCapCorrectCheckCameraChecked;		eRFID[22].bCapCorrectCapOn;eRFID[22].bCapCorrectNOK; eRFID[22].bFormPresent; eRFID[22].bBottlePresent; eRFID[22].bDosingTwoPhases; eRFID[22].nDispencerNr; eRFID[22].nDispencerNrSecondPhase; eRFID[22].lrDoseVolumeSV; eRFID[22].lrDoseVolumeCV; eRFID[22].lrDoseVolumeSVSecondPhase; eRFID[22].lrDoseVolumeCVSecondPhase; eRFID[22].bDosed;	eRFID[22].bDoseAborted; eRFID[22].bWeighed; eRFID[22].lrWeightSV; eRFID[22].lrWeightCV; eRFID[22].lrWeightMeasuredCV; eRFID[22].bWeightOK; eRFID[22].bCapPutted; eRFID[22].bCapChecked; eRFID[22].bCapOK; eRFID[22].bCapGripperScrewed; eRFID[22].bCapGripperScrewAborted; eRFID[22].bBottleTransferedToExit; eRFID[22].bBottleTransferedToLabeler; eRFID[22].lrWeightDif; eRFID[22].lrMinWeightCV;eRFID[22].lrMaxWeightCV;
eRFID[23].nCardNumber;eRFID[23].bCapCorrectChecked;	eRFID[23].bCapCorrectCheckCameraOK;		eRFID[23].bCapCorrectCheckCameraChecked;		eRFID[23].bCapCorrectCapOn;eRFID[23].bCapCorrectNOK; eRFID[23].bFormPresent; eRFID[23].bBottlePresent; eRFID[23].bDosingTwoPhases; eRFID[23].nDispencerNr; eRFID[23].nDispencerNrSecondPhase; eRFID[23].lrDoseVolumeSV; eRFID[23].lrDoseVolumeCV; eRFID[23].lrDoseVolumeSVSecondPhase; eRFID[23].lrDoseVolumeCVSecondPhase; eRFID[23].bDosed;	eRFID[23].bDoseAborted; eRFID[23].bWeighed; eRFID[23].lrWeightSV; eRFID[23].lrWeightCV; eRFID[23].lrWeightMeasuredCV; eRFID[23].bWeightOK; eRFID[23].bCapPutted; eRFID[23].bCapChecked; eRFID[23].bCapOK; eRFID[23].bCapGripperScrewed; eRFID[23].bCapGripperScrewAborted; eRFID[23].bBottleTransferedToExit; eRFID[23].bBottleTransferedToLabeler; eRFID[23].lrWeightDif; eRFID[23].lrMinWeightCV;eRFID[23].lrMaxWeightCV;
eRFID[24].nCardNumber;eRFID[24].bCapCorrectChecked;	eRFID[24].bCapCorrectCheckCameraOK;		eRFID[24].bCapCorrectCheckCameraChecked;		eRFID[24].bCapCorrectCapOn;eRFID[24].bCapCorrectNOK; eRFID[24].bFormPresent; eRFID[24].bBottlePresent; eRFID[24].bDosingTwoPhases; eRFID[24].nDispencerNr; eRFID[24].nDispencerNrSecondPhase; eRFID[24].lrDoseVolumeSV; eRFID[24].lrDoseVolumeCV; eRFID[24].lrDoseVolumeSVSecondPhase; eRFID[24].lrDoseVolumeCVSecondPhase; eRFID[24].bDosed;	eRFID[24].bDoseAborted; eRFID[24].bWeighed; eRFID[24].lrWeightSV; eRFID[24].lrWeightCV; eRFID[24].lrWeightMeasuredCV; eRFID[24].bWeightOK; eRFID[24].bCapPutted; eRFID[24].bCapChecked; eRFID[24].bCapOK; eRFID[24].bCapGripperScrewed; eRFID[24].bCapGripperScrewAborted; eRFID[24].bBottleTransferedToExit; eRFID[24].bBottleTransferedToLabeler; eRFID[24].lrWeightDif; eRFID[24].lrMinWeightCV;eRFID[24].lrMaxWeightCV;
eRFID[25].nCardNumber;eRFID[25].bCapCorrectChecked;	eRFID[25].bCapCorrectCheckCameraOK;		eRFID[25].bCapCorrectCheckCameraChecked;		eRFID[25].bCapCorrectCapOn;eRFID[25].bCapCorrectNOK; eRFID[25].bFormPresent; eRFID[25].bBottlePresent; eRFID[25].bDosingTwoPhases; eRFID[25].nDispencerNr; eRFID[25].nDispencerNrSecondPhase; eRFID[25].lrDoseVolumeSV; eRFID[25].lrDoseVolumeCV; eRFID[25].lrDoseVolumeSVSecondPhase; eRFID[25].lrDoseVolumeCVSecondPhase; eRFID[25].bDosed;	eRFID[25].bDoseAborted; eRFID[25].bWeighed; eRFID[25].lrWeightSV; eRFID[25].lrWeightCV; eRFID[25].lrWeightMeasuredCV; eRFID[25].bWeightOK; eRFID[25].bCapPutted; eRFID[25].bCapChecked; eRFID[25].bCapOK; eRFID[25].bCapGripperScrewed; eRFID[25].bCapGripperScrewAborted; eRFID[25].bBottleTransferedToExit; eRFID[25].bBottleTransferedToLabeler; eRFID[25].lrWeightDif; eRFID[25].lrMinWeightCV;eRFID[25].lrMaxWeightCV;
eRFID[26].nCardNumber;eRFID[26].bCapCorrectChecked;	eRFID[26].bCapCorrectCheckCameraOK;		eRFID[26].bCapCorrectCheckCameraChecked;		eRFID[26].bCapCorrectCapOn;eRFID[26].bCapCorrectNOK; eRFID[26].bFormPresent; eRFID[26].bBottlePresent; eRFID[26].bDosingTwoPhases; eRFID[26].nDispencerNr; eRFID[26].nDispencerNrSecondPhase; eRFID[26].lrDoseVolumeSV; eRFID[26].lrDoseVolumeCV; eRFID[26].lrDoseVolumeSVSecondPhase; eRFID[26].lrDoseVolumeCVSecondPhase; eRFID[26].bDosed;	eRFID[26].bDoseAborted; eRFID[26].bWeighed; eRFID[26].lrWeightSV; eRFID[26].lrWeightCV; eRFID[26].lrWeightMeasuredCV; eRFID[26].bWeightOK; eRFID[26].bCapPutted; eRFID[26].bCapChecked; eRFID[26].bCapOK; eRFID[26].bCapGripperScrewed; eRFID[26].bCapGripperScrewAborted; eRFID[26].bBottleTransferedToExit; eRFID[26].bBottleTransferedToLabeler; eRFID[26].lrWeightDif; eRFID[26].lrMinWeightCV;eRFID[26].lrMaxWeightCV;
eRFID[27].nCardNumber;eRFID[27].bCapCorrectChecked;	eRFID[27].bCapCorrectCheckCameraOK;		eRFID[27].bCapCorrectCheckCameraChecked;		eRFID[27].bCapCorrectCapOn;eRFID[27].bCapCorrectNOK; eRFID[27].bFormPresent; eRFID[27].bBottlePresent; eRFID[27].bDosingTwoPhases; eRFID[27].nDispencerNr; eRFID[27].nDispencerNrSecondPhase; eRFID[27].lrDoseVolumeSV; eRFID[27].lrDoseVolumeCV; eRFID[27].lrDoseVolumeSVSecondPhase; eRFID[27].lrDoseVolumeCVSecondPhase; eRFID[27].bDosed;	eRFID[27].bDoseAborted; eRFID[27].bWeighed; eRFID[27].lrWeightSV; eRFID[27].lrWeightCV; eRFID[27].lrWeightMeasuredCV; eRFID[27].bWeightOK; eRFID[27].bCapPutted; eRFID[27].bCapChecked; eRFID[27].bCapOK; eRFID[27].bCapGripperScrewed; eRFID[27].bCapGripperScrewAborted; eRFID[27].bBottleTransferedToExit; eRFID[27].bBottleTransferedToLabeler; eRFID[27].lrWeightDif; eRFID[27].lrMinWeightCV;eRFID[27].lrMaxWeightCV;
eRFID[28].nCardNumber;eRFID[28].bCapCorrectChecked;	eRFID[28].bCapCorrectCheckCameraOK;		eRFID[28].bCapCorrectCheckCameraChecked;		eRFID[28].bCapCorrectCapOn;eRFID[28].bCapCorrectNOK; eRFID[28].bFormPresent; eRFID[28].bBottlePresent; eRFID[28].bDosingTwoPhases; eRFID[28].nDispencerNr; eRFID[28].nDispencerNrSecondPhase; eRFID[28].lrDoseVolumeSV; eRFID[28].lrDoseVolumeCV; eRFID[28].lrDoseVolumeSVSecondPhase; eRFID[28].lrDoseVolumeCVSecondPhase; eRFID[28].bDosed;	eRFID[28].bDoseAborted; eRFID[28].bWeighed; eRFID[28].lrWeightSV; eRFID[28].lrWeightCV; eRFID[28].lrWeightMeasuredCV; eRFID[28].bWeightOK; eRFID[28].bCapPutted; eRFID[28].bCapChecked; eRFID[28].bCapOK; eRFID[28].bCapGripperScrewed; eRFID[28].bCapGripperScrewAborted; eRFID[28].bBottleTransferedToExit; eRFID[28].bBottleTransferedToLabeler; eRFID[28].lrWeightDif; eRFID[28].lrMinWeightCV;eRFID[28].lrMaxWeightCV;
eRFID[29].nCardNumber;eRFID[29].bCapCorrectChecked;	eRFID[29].bCapCorrectCheckCameraOK;		eRFID[29].bCapCorrectCheckCameraChecked;		eRFID[29].bCapCorrectCapOn;eRFID[29].bCapCorrectNOK; eRFID[29].bFormPresent; eRFID[29].bBottlePresent; eRFID[29].bDosingTwoPhases; eRFID[29].nDispencerNr; eRFID[29].nDispencerNrSecondPhase; eRFID[29].lrDoseVolumeSV; eRFID[29].lrDoseVolumeCV; eRFID[29].lrDoseVolumeSVSecondPhase; eRFID[29].lrDoseVolumeCVSecondPhase;	eRFID[29].bDosed;	eRFID[29].bDoseAborted; eRFID[29].bWeighed; eRFID[29].lrWeightSV; eRFID[29].lrWeightCV; eRFID[29].lrWeightMeasuredCV; eRFID[29].bWeightOK; eRFID[29].bCapPutted; eRFID[29].bCapChecked; eRFID[29].bCapOK; eRFID[29].bCapGripperScrewed; eRFID[29].bCapGripperScrewAborted; eRFID[29].bBottleTransferedToExit; eRFID[29].bBottleTransferedToLabeler; eRFID[29].lrWeightDif; eRFID[29].lrMinWeightCV;eRFID[29].lrMaxWeightCV;
eRFID[30].nCardNumber;eRFID[30].bCapCorrectChecked;	eRFID[30].bCapCorrectCheckCameraOK;		eRFID[30].bCapCorrectCheckCameraChecked;		eRFID[30].bCapCorrectCapOn;eRFID[30].bCapCorrectNOK; eRFID[30].bFormPresent; eRFID[30].bBottlePresent; eRFID[30].bDosingTwoPhases; eRFID[30].nDispencerNr; eRFID[30].nDispencerNrSecondPhase; eRFID[30].lrDoseVolumeSV; eRFID[30].lrDoseVolumeCV; eRFID[30].lrDoseVolumeSVSecondPhase; eRFID[30].lrDoseVolumeCVSecondPhase;	eRFID[30].bDosed;	eRFID[30].bDoseAborted; eRFID[30].bWeighed; eRFID[30].lrWeightSV; eRFID[30].lrWeightCV; eRFID[30].lrWeightMeasuredCV; eRFID[30].bWeightOK; eRFID[30].bCapPutted; eRFID[30].bCapChecked; eRFID[30].bCapOK; eRFID[30].bCapGripperScrewed; eRFID[30].bCapGripperScrewAborted; eRFID[30].bBottleTransferedToExit; eRFID[30].bBottleTransferedToLabeler; eRFID[30].lrWeightDif; eRFID[30].lrMinWeightCV;eRFID[30].lrMaxWeightCV;
eRFID[31].nCardNumber;eRFID[31].bCapCorrectChecked;	eRFID[31].bCapCorrectCheckCameraOK;		eRFID[31].bCapCorrectCheckCameraChecked;		eRFID[31].bCapCorrectCapOn;eRFID[31].bCapCorrectNOK; eRFID[31].bFormPresent; eRFID[31].bBottlePresent; eRFID[31].bDosingTwoPhases; eRFID[31].nDispencerNr; eRFID[31].nDispencerNrSecondPhase; eRFID[31].lrDoseVolumeSV; eRFID[31].lrDoseVolumeCV; eRFID[31].lrDoseVolumeSVSecondPhase; eRFID[31].lrDoseVolumeCVSecondPhase;	eRFID[31].bDosed;	eRFID[31].bDoseAborted; eRFID[31].bWeighed; eRFID[31].lrWeightSV; eRFID[31].lrWeightCV; eRFID[31].lrWeightMeasuredCV; eRFID[31].bWeightOK; eRFID[31].bCapPutted; eRFID[31].bCapChecked; eRFID[31].bCapOK; eRFID[31].bCapGripperScrewed; eRFID[31].bCapGripperScrewAborted; eRFID[31].bBottleTransferedToExit; eRFID[31].bBottleTransferedToLabeler; eRFID[31].lrWeightDif; eRFID[31].lrMinWeightCV;eRFID[31].lrMaxWeightCV;
eRFID[32].nCardNumber;eRFID[32].bCapCorrectChecked;	eRFID[32].bCapCorrectCheckCameraOK;		eRFID[32].bCapCorrectCheckCameraChecked;		eRFID[32].bCapCorrectCapOn;eRFID[32].bCapCorrectNOK; eRFID[32].bFormPresent; eRFID[32].bBottlePresent; eRFID[32].bDosingTwoPhases; eRFID[32].nDispencerNr; eRFID[32].nDispencerNrSecondPhase; eRFID[32].lrDoseVolumeSV; eRFID[32].lrDoseVolumeCV; eRFID[32].lrDoseVolumeSVSecondPhase; eRFID[32].lrDoseVolumeCVSecondPhase;	eRFID[32].bDosed;	eRFID[32].bDoseAborted; eRFID[32].bWeighed; eRFID[32].lrWeightSV; eRFID[32].lrWeightCV; eRFID[32].lrWeightMeasuredCV; eRFID[32].bWeightOK; eRFID[32].bCapPutted; eRFID[32].bCapChecked; eRFID[32].bCapOK; eRFID[32].bCapGripperScrewed; eRFID[32].bCapGripperScrewAborted; eRFID[32].bBottleTransferedToExit; eRFID[32].bBottleTransferedToLabeler; eRFID[32].lrWeightDif; eRFID[32].lrMinWeightCV;eRFID[32].lrMaxWeightCV;
eRFID[33].nCardNumber;eRFID[33].bCapCorrectChecked;	eRFID[33].bCapCorrectCheckCameraOK;		eRFID[33].bCapCorrectCheckCameraChecked;		eRFID[33].bCapCorrectCapOn;eRFID[33].bCapCorrectNOK; eRFID[33].bFormPresent; eRFID[33].bBottlePresent; eRFID[33].bDosingTwoPhases; eRFID[33].nDispencerNr; eRFID[33].nDispencerNrSecondPhase; eRFID[33].lrDoseVolumeSV; eRFID[33].lrDoseVolumeCV; eRFID[33].lrDoseVolumeSVSecondPhase; eRFID[33].lrDoseVolumeCVSecondPhase;	eRFID[33].bDosed;	eRFID[33].bDoseAborted; eRFID[33].bWeighed; eRFID[33].lrWeightSV; eRFID[33].lrWeightCV; eRFID[33].lrWeightMeasuredCV; eRFID[33].bWeightOK; eRFID[33].bCapPutted; eRFID[33].bCapChecked; eRFID[33].bCapOK; eRFID[33].bCapGripperScrewed; eRFID[33].bCapGripperScrewAborted; eRFID[33].bBottleTransferedToExit; eRFID[33].bBottleTransferedToLabeler; eRFID[33].lrWeightDif; eRFID[33].lrMinWeightCV;eRFID[33].lrMaxWeightCV;
eRFID[34].nCardNumber;eRFID[34].bCapCorrectChecked;	eRFID[34].bCapCorrectCheckCameraOK;		eRFID[34].bCapCorrectCheckCameraChecked;		eRFID[34].bCapCorrectCapOn;eRFID[34].bCapCorrectNOK; eRFID[34].bFormPresent; eRFID[34].bBottlePresent; eRFID[34].bDosingTwoPhases; eRFID[34].nDispencerNr; eRFID[34].nDispencerNrSecondPhase; eRFID[34].lrDoseVolumeSV; eRFID[34].lrDoseVolumeCV; eRFID[34].lrDoseVolumeSVSecondPhase; eRFID[34].lrDoseVolumeCVSecondPhase;	eRFID[34].bDosed;	eRFID[34].bDoseAborted; eRFID[34].bWeighed; eRFID[34].lrWeightSV; eRFID[34].lrWeightCV; eRFID[34].lrWeightMeasuredCV; eRFID[34].bWeightOK; eRFID[34].bCapPutted; eRFID[34].bCapChecked; eRFID[34].bCapOK; eRFID[34].bCapGripperScrewed; eRFID[34].bCapGripperScrewAborted; eRFID[34].bBottleTransferedToExit; eRFID[34].bBottleTransferedToLabeler; eRFID[34].lrWeightDif; eRFID[34].lrMinWeightCV;eRFID[34].lrMaxWeightCV;
eRFID[35].nCardNumber;eRFID[35].bCapCorrectChecked;	eRFID[35].bCapCorrectCheckCameraOK;		eRFID[35].bCapCorrectCheckCameraChecked;		eRFID[35].bCapCorrectCapOn;eRFID[35].bCapCorrectNOK; eRFID[35].bFormPresent; eRFID[35].bBottlePresent; eRFID[35].bDosingTwoPhases; eRFID[35].nDispencerNr; eRFID[35].nDispencerNrSecondPhase; eRFID[35].lrDoseVolumeSV; eRFID[35].lrDoseVolumeCV; eRFID[35].lrDoseVolumeSVSecondPhase; eRFID[35].lrDoseVolumeCVSecondPhase;	eRFID[35].bDosed;	eRFID[35].bDoseAborted; eRFID[35].bWeighed; eRFID[35].lrWeightSV; eRFID[35].lrWeightCV; eRFID[35].lrWeightMeasuredCV; eRFID[35].bWeightOK; eRFID[35].bCapPutted; eRFID[35].bCapChecked; eRFID[35].bCapOK; eRFID[35].bCapGripperScrewed; eRFID[35].bCapGripperScrewAborted; eRFID[35].bBottleTransferedToExit; eRFID[35].bBottleTransferedToLabeler; eRFID[35].lrWeightDif; eRFID[35].lrMinWeightCV;eRFID[35].lrMaxWeightCV;
eRFID[36].nCardNumber;eRFID[36].bCapCorrectChecked;	eRFID[36].bCapCorrectCheckCameraOK;		eRFID[36].bCapCorrectCheckCameraChecked;		eRFID[36].bCapCorrectCapOn;eRFID[36].bCapCorrectNOK; eRFID[36].bFormPresent; eRFID[36].bBottlePresent; eRFID[36].bDosingTwoPhases; eRFID[36].nDispencerNr; eRFID[36].nDispencerNrSecondPhase; eRFID[36].lrDoseVolumeSV; eRFID[36].lrDoseVolumeCV; eRFID[36].lrDoseVolumeSVSecondPhase; eRFID[36].lrDoseVolumeCVSecondPhase;	eRFID[36].bDosed;	eRFID[36].bDoseAborted; eRFID[36].bWeighed; eRFID[36].lrWeightSV; eRFID[36].lrWeightCV; eRFID[36].lrWeightMeasuredCV; eRFID[36].bWeightOK; eRFID[36].bCapPutted; eRFID[36].bCapChecked; eRFID[36].bCapOK; eRFID[36].bCapGripperScrewed; eRFID[36].bCapGripperScrewAborted; eRFID[36].bBottleTransferedToExit; eRFID[36].bBottleTransferedToLabeler; eRFID[36].lrWeightDif; eRFID[36].lrMinWeightCV;eRFID[36].lrMaxWeightCV;
eRFID[37].nCardNumber;eRFID[37].bCapCorrectChecked;	eRFID[37].bCapCorrectCheckCameraOK;		eRFID[37].bCapCorrectCheckCameraChecked;		eRFID[37].bCapCorrectCapOn;eRFID[37].bCapCorrectNOK; eRFID[37].bFormPresent; eRFID[37].bBottlePresent; eRFID[37].bDosingTwoPhases; eRFID[37].nDispencerNr; eRFID[37].nDispencerNrSecondPhase; eRFID[37].lrDoseVolumeSV; eRFID[37].lrDoseVolumeCV; eRFID[37].lrDoseVolumeSVSecondPhase; eRFID[37].lrDoseVolumeCVSecondPhase;	eRFID[37].bDosed;	eRFID[37].bDoseAborted; eRFID[37].bWeighed; eRFID[37].lrWeightSV; eRFID[37].lrWeightCV; eRFID[37].lrWeightMeasuredCV; eRFID[37].bWeightOK; eRFID[37].bCapPutted; eRFID[37].bCapChecked; eRFID[37].bCapOK; eRFID[37].bCapGripperScrewed; eRFID[37].bCapGripperScrewAborted; eRFID[37].bBottleTransferedToExit; eRFID[37].bBottleTransferedToLabeler; eRFID[37].lrWeightDif; eRFID[37].lrMinWeightCV;eRFID[37].lrMaxWeightCV;
eRFID[38].nCardNumber;eRFID[38].bCapCorrectChecked;	eRFID[38].bCapCorrectCheckCameraOK;		eRFID[38].bCapCorrectCheckCameraChecked;		eRFID[38].bCapCorrectCapOn;eRFID[38].bCapCorrectNOK; eRFID[38].bFormPresent; eRFID[38].bBottlePresent; eRFID[38].bDosingTwoPhases; eRFID[38].nDispencerNr; eRFID[38].nDispencerNrSecondPhase; eRFID[38].lrDoseVolumeSV; eRFID[38].lrDoseVolumeCV; eRFID[38].lrDoseVolumeSVSecondPhase; eRFID[38].lrDoseVolumeCVSecondPhase;	eRFID[38].bDosed;	eRFID[38].bDoseAborted; eRFID[38].bWeighed; eRFID[38].lrWeightSV; eRFID[38].lrWeightCV; eRFID[38].lrWeightMeasuredCV; eRFID[38].bWeightOK; eRFID[38].bCapPutted; eRFID[38].bCapChecked; eRFID[38].bCapOK; eRFID[38].bCapGripperScrewed; eRFID[38].bCapGripperScrewAborted; eRFID[38].bBottleTransferedToExit; eRFID[38].bBottleTransferedToLabeler; eRFID[38].lrWeightDif; eRFID[38].lrMinWeightCV;eRFID[38].lrMaxWeightCV;
eRFID[39].nCardNumber;eRFID[39].bCapCorrectChecked;	eRFID[39].bCapCorrectCheckCameraOK;		eRFID[39].bCapCorrectCheckCameraChecked;		eRFID[39].bCapCorrectCapOn;eRFID[39].bCapCorrectNOK; eRFID[39].bFormPresent; eRFID[39].bBottlePresent; eRFID[39].bDosingTwoPhases; eRFID[39].nDispencerNr; eRFID[39].nDispencerNrSecondPhase; eRFID[39].lrDoseVolumeSV; eRFID[39].lrDoseVolumeCV; eRFID[39].lrDoseVolumeSVSecondPhase; eRFID[39].lrDoseVolumeCVSecondPhase;	eRFID[39].bDosed;	eRFID[39].bDoseAborted; eRFID[39].bWeighed; eRFID[39].lrWeightSV; eRFID[39].lrWeightCV; eRFID[39].lrWeightMeasuredCV; eRFID[39].bWeightOK; eRFID[39].bCapPutted; eRFID[39].bCapChecked; eRFID[39].bCapOK; eRFID[39].bCapGripperScrewed; eRFID[39].bCapGripperScrewAborted; eRFID[39].bBottleTransferedToExit; eRFID[39].bBottleTransferedToLabeler; eRFID[39].lrWeightDif; eRFID[39].lrMinWeightCV;eRFID[39].lrMaxWeightCV;
eRFID[40].nCardNumber;eRFID[40].bCapCorrectChecked;	eRFID[40].bCapCorrectCheckCameraOK;		eRFID[40].bCapCorrectCheckCameraChecked;		eRFID[40].bCapCorrectCapOn;eRFID[40].bCapCorrectNOK; eRFID[40].bFormPresent; eRFID[40].bBottlePresent; eRFID[40].bDosingTwoPhases; eRFID[40].nDispencerNr; eRFID[40].nDispencerNrSecondPhase; eRFID[40].lrDoseVolumeSV; eRFID[40].lrDoseVolumeCV; eRFID[40].lrDoseVolumeSVSecondPhase; eRFID[40].lrDoseVolumeCVSecondPhase;	eRFID[40].bDosed;	eRFID[40].bDoseAborted; eRFID[40].bWeighed; eRFID[40].lrWeightSV; eRFID[40].lrWeightCV; eRFID[40].lrWeightMeasuredCV; eRFID[40].bWeightOK; eRFID[40].bCapPutted; eRFID[40].bCapChecked; eRFID[40].bCapOK; eRFID[40].bCapGripperScrewed; eRFID[40].bCapGripperScrewAborted; eRFID[40].bBottleTransferedToExit; eRFID[40].bBottleTransferedToLabeler; eRFID[40].lrWeightDif; eRFID[40].lrMinWeightCV;eRFID[40].lrMaxWeightCV;
eRFID[41].nCardNumber;eRFID[41].bCapCorrectChecked;	eRFID[41].bCapCorrectCheckCameraOK;		eRFID[41].bCapCorrectCheckCameraChecked;		eRFID[41].bCapCorrectCapOn;eRFID[41].bCapCorrectNOK; eRFID[41].bFormPresent; eRFID[41].bBottlePresent; eRFID[41].bDosingTwoPhases; eRFID[41].nDispencerNr; eRFID[41].nDispencerNrSecondPhase; eRFID[41].lrDoseVolumeSV; eRFID[41].lrDoseVolumeCV; eRFID[41].lrDoseVolumeSVSecondPhase; eRFID[41].lrDoseVolumeCVSecondPhase;	eRFID[41].bDosed;	eRFID[41].bDoseAborted; eRFID[41].bWeighed; eRFID[41].lrWeightSV; eRFID[41].lrWeightCV; eRFID[41].lrWeightMeasuredCV; eRFID[41].bWeightOK; eRFID[41].bCapPutted; eRFID[41].bCapChecked; eRFID[41].bCapOK; eRFID[41].bCapGripperScrewed; eRFID[41].bCapGripperScrewAborted; eRFID[41].bBottleTransferedToExit; eRFID[41].bBottleTransferedToLabeler; eRFID[41].lrWeightDif; eRFID[41].lrMinWeightCV;eRFID[41].lrMaxWeightCV;
eRFID[42].nCardNumber;eRFID[42].bCapCorrectChecked;	eRFID[42].bCapCorrectCheckCameraOK;		eRFID[42].bCapCorrectCheckCameraChecked;		eRFID[42].bCapCorrectCapOn;eRFID[42].bCapCorrectNOK; eRFID[42].bFormPresent; eRFID[42].bBottlePresent; eRFID[42].bDosingTwoPhases; eRFID[42].nDispencerNr; eRFID[42].nDispencerNrSecondPhase; eRFID[42].lrDoseVolumeSV; eRFID[42].lrDoseVolumeCV; eRFID[42].lrDoseVolumeSVSecondPhase; eRFID[42].lrDoseVolumeCVSecondPhase;	eRFID[42].bDosed;	eRFID[42].bDoseAborted; eRFID[42].bWeighed; eRFID[42].lrWeightSV; eRFID[42].lrWeightCV; eRFID[42].lrWeightMeasuredCV; eRFID[42].bWeightOK; eRFID[42].bCapPutted; eRFID[42].bCapChecked; eRFID[42].bCapOK; eRFID[42].bCapGripperScrewed; eRFID[42].bCapGripperScrewAborted; eRFID[42].bBottleTransferedToExit; eRFID[42].bBottleTransferedToLabeler; eRFID[42].lrWeightDif; eRFID[42].lrMinWeightCV;eRFID[42].lrMaxWeightCV;
eRFID[43].nCardNumber;eRFID[43].bCapCorrectChecked;	eRFID[43].bCapCorrectCheckCameraOK;		eRFID[43].bCapCorrectCheckCameraChecked;		eRFID[43].bCapCorrectCapOn;eRFID[43].bCapCorrectNOK; eRFID[43].bFormPresent; eRFID[43].bBottlePresent; eRFID[43].bDosingTwoPhases; eRFID[43].nDispencerNr; eRFID[43].nDispencerNrSecondPhase; eRFID[43].lrDoseVolumeSV; eRFID[43].lrDoseVolumeCV; eRFID[43].lrDoseVolumeSVSecondPhase; eRFID[43].lrDoseVolumeCVSecondPhase;	eRFID[43].bDosed;	eRFID[43].bDoseAborted; eRFID[43].bWeighed; eRFID[43].lrWeightSV; eRFID[43].lrWeightCV; eRFID[43].lrWeightMeasuredCV; eRFID[43].bWeightOK; eRFID[43].bCapPutted; eRFID[43].bCapChecked; eRFID[43].bCapOK; eRFID[43].bCapGripperScrewed; eRFID[43].bCapGripperScrewAborted; eRFID[43].bBottleTransferedToExit; eRFID[43].bBottleTransferedToLabeler; eRFID[43].lrWeightDif; eRFID[43].lrMinWeightCV;eRFID[43].lrMaxWeightCV;
eRFID[44].nCardNumber;eRFID[44].bCapCorrectChecked;	eRFID[44].bCapCorrectCheckCameraOK;		eRFID[44].bCapCorrectCheckCameraChecked;		eRFID[44].bCapCorrectCapOn;eRFID[44].bCapCorrectNOK; eRFID[44].bFormPresent; eRFID[44].bBottlePresent; eRFID[44].bDosingTwoPhases; eRFID[44].nDispencerNr; eRFID[44].nDispencerNrSecondPhase; eRFID[44].lrDoseVolumeSV; eRFID[44].lrDoseVolumeCV; eRFID[44].lrDoseVolumeSVSecondPhase; eRFID[44].lrDoseVolumeCVSecondPhase;	eRFID[44].bDosed;	eRFID[44].bDoseAborted; eRFID[44].bWeighed; eRFID[44].lrWeightSV; eRFID[44].lrWeightCV; eRFID[44].lrWeightMeasuredCV; eRFID[44].bWeightOK; eRFID[44].bCapPutted; eRFID[44].bCapChecked; eRFID[44].bCapOK; eRFID[44].bCapGripperScrewed; eRFID[44].bCapGripperScrewAborted; eRFID[44].bBottleTransferedToExit; eRFID[44].bBottleTransferedToLabeler; eRFID[44].lrWeightDif; eRFID[44].lrMinWeightCV;eRFID[44].lrMaxWeightCV;
eRFID[45].nCardNumber;eRFID[45].bCapCorrectChecked;	eRFID[45].bCapCorrectCheckCameraOK;		eRFID[45].bCapCorrectCheckCameraChecked;		eRFID[45].bCapCorrectCapOn;eRFID[45].bCapCorrectNOK; eRFID[45].bFormPresent; eRFID[45].bBottlePresent; eRFID[45].bDosingTwoPhases; eRFID[45].nDispencerNr; eRFID[45].nDispencerNrSecondPhase; eRFID[45].lrDoseVolumeSV; eRFID[45].lrDoseVolumeCV; eRFID[45].lrDoseVolumeSVSecondPhase; eRFID[45].lrDoseVolumeCVSecondPhase;	eRFID[45].bDosed;	eRFID[45].bDoseAborted; eRFID[45].bWeighed; eRFID[45].lrWeightSV; eRFID[45].lrWeightCV; eRFID[45].lrWeightMeasuredCV; eRFID[45].bWeightOK; eRFID[45].bCapPutted; eRFID[45].bCapChecked; eRFID[45].bCapOK; eRFID[45].bCapGripperScrewed; eRFID[45].bCapGripperScrewAborted; eRFID[45].bBottleTransferedToExit; eRFID[45].bBottleTransferedToLabeler; eRFID[45].lrWeightDif; eRFID[45].lrMinWeightCV;eRFID[45].lrMaxWeightCV;
eRFID[46].nCardNumber;eRFID[46].bCapCorrectChecked;	eRFID[46].bCapCorrectCheckCameraOK;		eRFID[46].bCapCorrectCheckCameraChecked;		eRFID[46].bCapCorrectCapOn;eRFID[46].bCapCorrectNOK; eRFID[46].bFormPresent; eRFID[46].bBottlePresent; eRFID[46].bDosingTwoPhases; eRFID[46].nDispencerNr; eRFID[46].nDispencerNrSecondPhase; eRFID[46].lrDoseVolumeSV; eRFID[46].lrDoseVolumeCV; eRFID[46].lrDoseVolumeSVSecondPhase; eRFID[46].lrDoseVolumeCVSecondPhase;	eRFID[46].bDosed;	eRFID[46].bDoseAborted; eRFID[46].bWeighed; eRFID[46].lrWeightSV; eRFID[46].lrWeightCV; eRFID[46].lrWeightMeasuredCV; eRFID[46].bWeightOK; eRFID[46].bCapPutted; eRFID[46].bCapChecked; eRFID[46].bCapOK; eRFID[46].bCapGripperScrewed; eRFID[46].bCapGripperScrewAborted; eRFID[46].bBottleTransferedToExit; eRFID[46].bBottleTransferedToLabeler; eRFID[46].lrWeightDif; eRFID[46].lrMinWeightCV;eRFID[46].lrMaxWeightCV;
eRFID[47].nCardNumber;eRFID[47].bCapCorrectChecked;	eRFID[47].bCapCorrectCheckCameraOK;		eRFID[47].bCapCorrectCheckCameraChecked;		eRFID[47].bCapCorrectCapOn;eRFID[47].bCapCorrectNOK; eRFID[47].bFormPresent; eRFID[47].bBottlePresent; eRFID[47].bDosingTwoPhases; eRFID[47].nDispencerNr; eRFID[47].nDispencerNrSecondPhase; eRFID[47].lrDoseVolumeSV; eRFID[47].lrDoseVolumeCV; eRFID[47].lrDoseVolumeSVSecondPhase; eRFID[47].lrDoseVolumeCVSecondPhase;	eRFID[47].bDosed;	eRFID[47].bDoseAborted; eRFID[47].bWeighed; eRFID[47].lrWeightSV; eRFID[47].lrWeightCV; eRFID[47].lrWeightMeasuredCV; eRFID[47].bWeightOK; eRFID[47].bCapPutted; eRFID[47].bCapChecked; eRFID[47].bCapOK; eRFID[47].bCapGripperScrewed; eRFID[47].bCapGripperScrewAborted; eRFID[47].bBottleTransferedToExit; eRFID[47].bBottleTransferedToLabeler; eRFID[47].lrWeightDif; eRFID[47].lrMinWeightCV;eRFID[47].lrMaxWeightCV;
eRFID[48].nCardNumber;eRFID[48].bCapCorrectChecked;	eRFID[48].bCapCorrectCheckCameraOK;		eRFID[48].bCapCorrectCheckCameraChecked;		eRFID[48].bCapCorrectCapOn;eRFID[48].bCapCorrectNOK; eRFID[48].bFormPresent; eRFID[48].bBottlePresent; eRFID[48].bDosingTwoPhases; eRFID[48].nDispencerNr; eRFID[48].nDispencerNrSecondPhase; eRFID[48].lrDoseVolumeSV; eRFID[48].lrDoseVolumeCV; eRFID[48].lrDoseVolumeSVSecondPhase; eRFID[48].lrDoseVolumeCVSecondPhase;	eRFID[48].bDosed;	eRFID[48].bDoseAborted; eRFID[48].bWeighed; eRFID[48].lrWeightSV; eRFID[48].lrWeightCV; eRFID[48].lrWeightMeasuredCV; eRFID[48].bWeightOK; eRFID[48].bCapPutted; eRFID[48].bCapChecked; eRFID[48].bCapOK; eRFID[48].bCapGripperScrewed; eRFID[48].bCapGripperScrewAborted; eRFID[48].bBottleTransferedToExit; eRFID[48].bBottleTransferedToLabeler; eRFID[48].lrWeightDif; eRFID[48].lrMinWeightCV;eRFID[48].lrMaxWeightCV;
eRFID[49].nCardNumber;eRFID[49].bCapCorrectChecked;	eRFID[49].bCapCorrectCheckCameraOK;		eRFID[49].bCapCorrectCheckCameraChecked;		eRFID[49].bCapCorrectCapOn;eRFID[49].bCapCorrectNOK; eRFID[49].bFormPresent; eRFID[49].bBottlePresent; eRFID[49].bDosingTwoPhases; eRFID[49].nDispencerNr; eRFID[49].nDispencerNrSecondPhase; eRFID[49].lrDoseVolumeSV; eRFID[49].lrDoseVolumeCV; eRFID[49].lrDoseVolumeSVSecondPhase; eRFID[49].lrDoseVolumeCVSecondPhase;	eRFID[49].bDosed;	eRFID[49].bDoseAborted; eRFID[49].bWeighed; eRFID[49].lrWeightSV; eRFID[49].lrWeightCV; eRFID[49].lrWeightMeasuredCV; eRFID[49].bWeightOK; eRFID[49].bCapPutted; eRFID[49].bCapChecked; eRFID[49].bCapOK; eRFID[49].bCapGripperScrewed; eRFID[49].bCapGripperScrewAborted; eRFID[49].bBottleTransferedToExit; eRFID[49].bBottleTransferedToLabeler; eRFID[49].lrWeightDif; eRFID[49].lrMinWeightCV;eRFID[49].lrMaxWeightCV;
eRFID[50].nCardNumber;eRFID[50].bCapCorrectChecked;	eRFID[50].bCapCorrectCheckCameraOK;		eRFID[50].bCapCorrectCheckCameraChecked;		eRFID[50].bCapCorrectCapOn;eRFID[50].bCapCorrectNOK; eRFID[50].bFormPresent; eRFID[50].bBottlePresent; eRFID[50].bDosingTwoPhases; eRFID[50].nDispencerNr; eRFID[50].nDispencerNrSecondPhase; eRFID[50].lrDoseVolumeSV; eRFID[50].lrDoseVolumeCV; eRFID[50].lrDoseVolumeSVSecondPhase; eRFID[50].lrDoseVolumeCVSecondPhase;	eRFID[50].bDosed;	eRFID[50].bDoseAborted; eRFID[50].bWeighed; eRFID[50].lrWeightSV; eRFID[50].lrWeightCV; eRFID[50].lrWeightMeasuredCV; eRFID[50].bWeightOK; eRFID[50].bCapPutted; eRFID[50].bCapChecked; eRFID[50].bCapOK; eRFID[50].bCapGripperScrewed; eRFID[50].bCapGripperScrewAborted; eRFID[50].bBottleTransferedToExit; eRFID[50].bBottleTransferedToLabeler; eRFID[50].lrWeightDif; eRFID[50].lrMinWeightCV;eRFID[50].lrMaxWeightCV;
eRFID[51].nCardNumber;eRFID[51].bCapCorrectChecked;	eRFID[51].bCapCorrectCheckCameraOK;		eRFID[51].bCapCorrectCheckCameraChecked;		eRFID[51].bCapCorrectCapOn;eRFID[51].bCapCorrectNOK; eRFID[51].bFormPresent; eRFID[51].bBottlePresent; eRFID[51].bDosingTwoPhases; eRFID[51].nDispencerNr; eRFID[51].nDispencerNrSecondPhase; eRFID[51].lrDoseVolumeSV; eRFID[51].lrDoseVolumeCV; eRFID[51].lrDoseVolumeSVSecondPhase; eRFID[51].lrDoseVolumeCVSecondPhase;	eRFID[51].bDosed;	eRFID[51].bDoseAborted; eRFID[51].bWeighed; eRFID[51].lrWeightSV; eRFID[51].lrWeightCV; eRFID[51].lrWeightMeasuredCV; eRFID[51].bWeightOK; eRFID[51].bCapPutted; eRFID[51].bCapChecked; eRFID[51].bCapOK; eRFID[51].bCapGripperScrewed; eRFID[51].bCapGripperScrewAborted; eRFID[51].bBottleTransferedToExit; eRFID[51].bBottleTransferedToLabeler; eRFID[51].lrWeightDif; eRFID[51].lrMinWeightCV;eRFID[51].lrMaxWeightCV;
eRFID[52].nCardNumber;eRFID[52].bCapCorrectChecked;	eRFID[52].bCapCorrectCheckCameraOK;		eRFID[52].bCapCorrectCheckCameraChecked;		eRFID[52].bCapCorrectCapOn;eRFID[52].bCapCorrectNOK; eRFID[52].bFormPresent; eRFID[52].bBottlePresent; eRFID[52].bDosingTwoPhases; eRFID[52].nDispencerNr; eRFID[52].nDispencerNrSecondPhase; eRFID[52].lrDoseVolumeSV; eRFID[52].lrDoseVolumeCV; eRFID[52].lrDoseVolumeSVSecondPhase; eRFID[52].lrDoseVolumeCVSecondPhase;	eRFID[52].bDosed;	eRFID[52].bDoseAborted; eRFID[52].bWeighed; eRFID[52].lrWeightSV; eRFID[52].lrWeightCV; eRFID[52].lrWeightMeasuredCV; eRFID[52].bWeightOK; eRFID[52].bCapPutted; eRFID[52].bCapChecked; eRFID[52].bCapOK; eRFID[52].bCapGripperScrewed; eRFID[52].bCapGripperScrewAborted; eRFID[52].bBottleTransferedToExit; eRFID[52].bBottleTransferedToLabeler; eRFID[52].lrWeightDif; eRFID[52].lrMinWeightCV;eRFID[52].lrMaxWeightCV;
eRFID[53].nCardNumber;eRFID[53].bCapCorrectChecked;	eRFID[53].bCapCorrectCheckCameraOK;		eRFID[53].bCapCorrectCheckCameraChecked;		eRFID[53].bCapCorrectCapOn;eRFID[53].bCapCorrectNOK; eRFID[53].bFormPresent; eRFID[53].bBottlePresent; eRFID[53].bDosingTwoPhases; eRFID[53].nDispencerNr; eRFID[53].nDispencerNrSecondPhase; eRFID[53].lrDoseVolumeSV; eRFID[53].lrDoseVolumeCV; eRFID[53].lrDoseVolumeSVSecondPhase; eRFID[53].lrDoseVolumeCVSecondPhase; eRFID[53].bDosed;	eRFID[53].bDoseAborted; eRFID[53].bWeighed; eRFID[53].lrWeightSV; eRFID[53].lrWeightCV; eRFID[53].lrWeightMeasuredCV; eRFID[53].bWeightOK; eRFID[53].bCapPutted; eRFID[53].bCapChecked; eRFID[53].bCapOK; eRFID[53].bCapGripperScrewed; eRFID[53].bCapGripperScrewAborted; eRFID[53].bBottleTransferedToExit; eRFID[53].bBottleTransferedToLabeler; eRFID[53].lrWeightDif; eRFID[53].lrMinWeightCV;eRFID[53].lrMaxWeightCV;
eRFID[54].nCardNumber;eRFID[54].bCapCorrectChecked;	eRFID[54].bCapCorrectCheckCameraOK;		eRFID[54].bCapCorrectCheckCameraChecked;		eRFID[54].bCapCorrectCapOn;eRFID[54].bCapCorrectNOK; eRFID[54].bFormPresent; eRFID[54].bBottlePresent; eRFID[54].bDosingTwoPhases; eRFID[54].nDispencerNr; eRFID[54].nDispencerNrSecondPhase; eRFID[54].lrDoseVolumeSV; eRFID[54].lrDoseVolumeCV; eRFID[54].lrDoseVolumeSVSecondPhase; eRFID[54].lrDoseVolumeCVSecondPhase; eRFID[54].bDosed;	eRFID[54].bDoseAborted; eRFID[54].bWeighed; eRFID[54].lrWeightSV; eRFID[54].lrWeightCV; eRFID[54].lrWeightMeasuredCV; eRFID[54].bWeightOK; eRFID[54].bCapPutted; eRFID[54].bCapChecked; eRFID[54].bCapOK; eRFID[54].bCapGripperScrewed; eRFID[54].bCapGripperScrewAborted; eRFID[54].bBottleTransferedToExit; eRFID[54].bBottleTransferedToLabeler; eRFID[54].lrWeightDif; eRFID[54].lrMinWeightCV;eRFID[54].lrMaxWeightCV;
eRFID[55].nCardNumber;eRFID[55].bCapCorrectChecked;	eRFID[55].bCapCorrectCheckCameraOK;		eRFID[55].bCapCorrectCheckCameraChecked;		eRFID[55].bCapCorrectCapOn;eRFID[55].bCapCorrectNOK; eRFID[55].bFormPresent; eRFID[55].bBottlePresent; eRFID[55].bDosingTwoPhases; eRFID[55].nDispencerNr; eRFID[55].nDispencerNrSecondPhase; eRFID[55].lrDoseVolumeSV; eRFID[55].lrDoseVolumeCV; eRFID[55].lrDoseVolumeSVSecondPhase; eRFID[55].lrDoseVolumeCVSecondPhase; eRFID[55].bDosed;	eRFID[55].bDoseAborted; eRFID[55].bWeighed; eRFID[55].lrWeightSV; eRFID[55].lrWeightCV; eRFID[55].lrWeightMeasuredCV; eRFID[55].bWeightOK; eRFID[55].bCapPutted; eRFID[55].bCapChecked; eRFID[55].bCapOK; eRFID[55].bCapGripperScrewed; eRFID[55].bCapGripperScrewAborted; eRFID[55].bBottleTransferedToExit; eRFID[55].bBottleTransferedToLabeler; eRFID[55].lrWeightDif; eRFID[55].lrMinWeightCV;eRFID[55].lrMaxWeightCV;
eRFID[56].nCardNumber;eRFID[56].bCapCorrectChecked;	eRFID[56].bCapCorrectCheckCameraOK;		eRFID[56].bCapCorrectCheckCameraChecked;		eRFID[56].bCapCorrectCapOn;eRFID[56].bCapCorrectNOK; eRFID[56].bFormPresent; eRFID[56].bBottlePresent; eRFID[56].bDosingTwoPhases; eRFID[56].nDispencerNr; eRFID[56].nDispencerNrSecondPhase; eRFID[56].lrDoseVolumeSV; eRFID[56].lrDoseVolumeCV; eRFID[56].lrDoseVolumeSVSecondPhase; eRFID[56].lrDoseVolumeCVSecondPhase; eRFID[56].bDosed;	eRFID[56].bDoseAborted; eRFID[56].bWeighed; eRFID[56].lrWeightSV; eRFID[56].lrWeightCV; eRFID[56].lrWeightMeasuredCV; eRFID[56].bWeightOK; eRFID[56].bCapPutted; eRFID[56].bCapChecked; eRFID[56].bCapOK; eRFID[56].bCapGripperScrewed; eRFID[56].bCapGripperScrewAborted; eRFID[56].bBottleTransferedToExit; eRFID[56].bBottleTransferedToLabeler; eRFID[56].lrWeightDif; eRFID[56].lrMinWeightCV;eRFID[56].lrMaxWeightCV;
eRFID[57].nCardNumber;eRFID[57].bCapCorrectChecked;	eRFID[57].bCapCorrectCheckCameraOK;		eRFID[57].bCapCorrectCheckCameraChecked;		eRFID[57].bCapCorrectCapOn;eRFID[57].bCapCorrectNOK; eRFID[57].bFormPresent; eRFID[57].bBottlePresent; eRFID[57].bDosingTwoPhases; eRFID[57].nDispencerNr; eRFID[57].nDispencerNrSecondPhase; eRFID[57].lrDoseVolumeSV; eRFID[57].lrDoseVolumeCV; eRFID[57].lrDoseVolumeSVSecondPhase; eRFID[57].lrDoseVolumeCVSecondPhase; eRFID[57].bDosed;	eRFID[57].bDoseAborted; eRFID[57].bWeighed; eRFID[57].lrWeightSV; eRFID[57].lrWeightCV; eRFID[57].lrWeightMeasuredCV; eRFID[57].bWeightOK; eRFID[57].bCapPutted; eRFID[57].bCapChecked; eRFID[57].bCapOK; eRFID[57].bCapGripperScrewed; eRFID[57].bCapGripperScrewAborted; eRFID[57].bBottleTransferedToExit; eRFID[57].bBottleTransferedToLabeler; eRFID[57].lrWeightDif; eRFID[57].lrMinWeightCV;eRFID[57].lrMaxWeightCV;
eRFID[58].nCardNumber;eRFID[58].bCapCorrectChecked;	eRFID[58].bCapCorrectCheckCameraOK;		eRFID[58].bCapCorrectCheckCameraChecked;		eRFID[58].bCapCorrectCapOn;eRFID[58].bCapCorrectNOK; eRFID[58].bFormPresent; eRFID[58].bBottlePresent; eRFID[58].bDosingTwoPhases; eRFID[58].nDispencerNr; eRFID[58].nDispencerNrSecondPhase; eRFID[58].lrDoseVolumeSV; eRFID[58].lrDoseVolumeCV; eRFID[58].lrDoseVolumeSVSecondPhase; eRFID[58].lrDoseVolumeCVSecondPhase; eRFID[58].bDosed;	eRFID[58].bDoseAborted; eRFID[58].bWeighed; eRFID[58].lrWeightSV; eRFID[58].lrWeightCV; eRFID[58].lrWeightMeasuredCV; eRFID[58].bWeightOK; eRFID[58].bCapPutted; eRFID[58].bCapChecked; eRFID[58].bCapOK; eRFID[58].bCapGripperScrewed; eRFID[58].bCapGripperScrewAborted; eRFID[58].bBottleTransferedToExit; eRFID[58].bBottleTransferedToLabeler; eRFID[58].lrWeightDif; eRFID[58].lrMinWeightCV;eRFID[58].lrMaxWeightCV;
eRFID[59].nCardNumber;eRFID[59].bCapCorrectChecked;	eRFID[59].bCapCorrectCheckCameraOK;		eRFID[59].bCapCorrectCheckCameraChecked;		eRFID[59].bCapCorrectCapOn;eRFID[59].bCapCorrectNOK; eRFID[59].bFormPresent; eRFID[59].bBottlePresent; eRFID[59].bDosingTwoPhases; eRFID[59].nDispencerNr; eRFID[59].nDispencerNrSecondPhase; eRFID[59].lrDoseVolumeSV; eRFID[59].lrDoseVolumeCV; eRFID[59].lrDoseVolumeSVSecondPhase; eRFID[59].lrDoseVolumeCVSecondPhase; eRFID[59].bDosed;	eRFID[59].bDoseAborted; eRFID[59].bWeighed; eRFID[59].lrWeightSV; eRFID[59].lrWeightCV; eRFID[59].lrWeightMeasuredCV; eRFID[59].bWeightOK; eRFID[59].bCapPutted; eRFID[59].bCapChecked; eRFID[59].bCapOK; eRFID[59].bCapGripperScrewed; eRFID[59].bCapGripperScrewAborted; eRFID[59].bBottleTransferedToExit; eRFID[59].bBottleTransferedToLabeler; eRFID[59].lrWeightDif; eRFID[59].lrMinWeightCV;eRFID[59].lrMaxWeightCV;
eRFID[60].nCardNumber;eRFID[60].bCapCorrectChecked;	eRFID[60].bCapCorrectCheckCameraOK;		eRFID[60].bCapCorrectCheckCameraChecked;		eRFID[60].bCapCorrectCapOn;eRFID[60].bCapCorrectNOK; eRFID[60].bFormPresent; eRFID[60].bBottlePresent; eRFID[60].bDosingTwoPhases; eRFID[60].nDispencerNr; eRFID[60].nDispencerNrSecondPhase; eRFID[60].lrDoseVolumeSV; eRFID[60].lrDoseVolumeCV; eRFID[60].lrDoseVolumeSVSecondPhase; eRFID[60].lrDoseVolumeCVSecondPhase; eRFID[60].bDosed;	eRFID[60].bDoseAborted; eRFID[60].bWeighed; eRFID[60].lrWeightSV; eRFID[60].lrWeightCV; eRFID[60].lrWeightMeasuredCV; eRFID[60].bWeightOK; eRFID[60].bCapPutted; eRFID[60].bCapChecked; eRFID[60].bCapOK; eRFID[60].bCapGripperScrewed; eRFID[60].bCapGripperScrewAborted; eRFID[60].bBottleTransferedToExit; eRFID[60].bBottleTransferedToLabeler; eRFID[60].lrWeightDif; eRFID[60].lrMinWeightCV;eRFID[60].lrMaxWeightCV;
eRFID[61].nCardNumber;eRFID[61].bCapCorrectChecked;	eRFID[61].bCapCorrectCheckCameraOK;		eRFID[61].bCapCorrectCheckCameraChecked;		eRFID[61].bCapCorrectCapOn;eRFID[61].bCapCorrectNOK; eRFID[61].bFormPresent; eRFID[61].bBottlePresent; eRFID[61].bDosingTwoPhases; eRFID[61].nDispencerNr; eRFID[61].nDispencerNrSecondPhase; eRFID[61].lrDoseVolumeSV; eRFID[61].lrDoseVolumeCV; eRFID[61].lrDoseVolumeSVSecondPhase; eRFID[61].lrDoseVolumeCVSecondPhase; eRFID[61].bDosed;	eRFID[61].bDoseAborted; eRFID[61].bWeighed; eRFID[61].lrWeightSV; eRFID[61].lrWeightCV; eRFID[61].lrWeightMeasuredCV; eRFID[61].bWeightOK; eRFID[61].bCapPutted; eRFID[61].bCapChecked; eRFID[61].bCapOK; eRFID[61].bCapGripperScrewed; eRFID[61].bCapGripperScrewAborted; eRFID[61].bBottleTransferedToExit; eRFID[61].bBottleTransferedToLabeler; eRFID[61].lrWeightDif; eRFID[61].lrMinWeightCV;eRFID[61].lrMaxWeightCV;
eRFID[62].nCardNumber;eRFID[62].bCapCorrectChecked;	eRFID[62].bCapCorrectCheckCameraOK;		eRFID[62].bCapCorrectCheckCameraChecked;		eRFID[62].bCapCorrectCapOn;eRFID[62].bCapCorrectNOK; eRFID[62].bFormPresent; eRFID[62].bBottlePresent; eRFID[62].bDosingTwoPhases; eRFID[62].nDispencerNr; eRFID[62].nDispencerNrSecondPhase; eRFID[62].lrDoseVolumeSV; eRFID[62].lrDoseVolumeCV; eRFID[62].lrDoseVolumeSVSecondPhase; eRFID[62].lrDoseVolumeCVSecondPhase; eRFID[62].bDosed;	eRFID[62].bDoseAborted; eRFID[62].bWeighed; eRFID[62].lrWeightSV; eRFID[62].lrWeightCV; eRFID[62].lrWeightMeasuredCV; eRFID[62].bWeightOK; eRFID[62].bCapPutted; eRFID[62].bCapChecked; eRFID[62].bCapOK; eRFID[62].bCapGripperScrewed; eRFID[62].bCapGripperScrewAborted; eRFID[62].bBottleTransferedToExit; eRFID[62].bBottleTransferedToLabeler; eRFID[62].lrWeightDif; eRFID[62].lrMinWeightCV;eRFID[62].lrMaxWeightCV;
eRFID[63].nCardNumber;eRFID[63].bCapCorrectChecked;	eRFID[63].bCapCorrectCheckCameraOK;		eRFID[63].bCapCorrectCheckCameraChecked;		eRFID[63].bCapCorrectCapOn;eRFID[63].bCapCorrectNOK; eRFID[63].bFormPresent; eRFID[63].bBottlePresent; eRFID[63].bDosingTwoPhases; eRFID[63].nDispencerNr; eRFID[63].nDispencerNrSecondPhase; eRFID[63].lrDoseVolumeSV; eRFID[63].lrDoseVolumeCV; eRFID[63].lrDoseVolumeSVSecondPhase; eRFID[63].lrDoseVolumeCVSecondPhase; eRFID[63].bDosed;	eRFID[63].bDoseAborted; eRFID[63].bWeighed; eRFID[63].lrWeightSV; eRFID[63].lrWeightCV; eRFID[63].lrWeightMeasuredCV; eRFID[63].bWeightOK; eRFID[63].bCapPutted; eRFID[63].bCapChecked; eRFID[63].bCapOK; eRFID[63].bCapGripperScrewed; eRFID[63].bCapGripperScrewAborted; eRFID[63].bBottleTransferedToExit; eRFID[63].bBottleTransferedToLabeler; eRFID[63].lrWeightDif; eRFID[63].lrMinWeightCV;eRFID[63].lrMaxWeightCV;
eRFID[64].nCardNumber;eRFID[64].bCapCorrectChecked;	eRFID[64].bCapCorrectCheckCameraOK;		eRFID[64].bCapCorrectCheckCameraChecked;		eRFID[64].bCapCorrectCapOn;eRFID[64].bCapCorrectNOK; eRFID[64].bFormPresent; eRFID[64].bBottlePresent; eRFID[64].bDosingTwoPhases; eRFID[64].nDispencerNr; eRFID[64].nDispencerNrSecondPhase; eRFID[64].lrDoseVolumeSV; eRFID[64].lrDoseVolumeCV; eRFID[64].lrDoseVolumeSVSecondPhase; eRFID[64].lrDoseVolumeCVSecondPhase; eRFID[64].bDosed;	eRFID[64].bDoseAborted; eRFID[64].bWeighed; eRFID[64].lrWeightSV; eRFID[64].lrWeightCV; eRFID[64].lrWeightMeasuredCV; eRFID[64].bWeightOK; eRFID[64].bCapPutted; eRFID[64].bCapChecked; eRFID[64].bCapOK; eRFID[64].bCapGripperScrewed; eRFID[64].bCapGripperScrewAborted; eRFID[64].bBottleTransferedToExit; eRFID[64].bBottleTransferedToLabeler; eRFID[64].lrWeightDif; eRFID[64].lrMinWeightCV;eRFID[64].lrMaxWeightCV;
eRFID[65].nCardNumber;eRFID[65].bCapCorrectChecked;	eRFID[65].bCapCorrectCheckCameraOK;		eRFID[65].bCapCorrectCheckCameraChecked;		eRFID[65].bCapCorrectCapOn;eRFID[65].bCapCorrectNOK; eRFID[65].bFormPresent; eRFID[65].bBottlePresent; eRFID[65].bDosingTwoPhases; eRFID[65].nDispencerNr; eRFID[65].nDispencerNrSecondPhase; eRFID[65].lrDoseVolumeSV; eRFID[65].lrDoseVolumeCV; eRFID[65].lrDoseVolumeSVSecondPhase; eRFID[65].lrDoseVolumeCVSecondPhase; eRFID[65].bDosed;	eRFID[65].bDoseAborted; eRFID[65].bWeighed; eRFID[65].lrWeightSV; eRFID[65].lrWeightCV; eRFID[65].lrWeightMeasuredCV; eRFID[65].bWeightOK; eRFID[65].bCapPutted; eRFID[65].bCapChecked; eRFID[65].bCapOK; eRFID[65].bCapGripperScrewed; eRFID[65].bCapGripperScrewAborted; eRFID[65].bBottleTransferedToExit; eRFID[65].bBottleTransferedToLabeler; eRFID[65].lrWeightDif; eRFID[65].lrMinWeightCV;eRFID[65].lrMaxWeightCV;
eRFID[66].nCardNumber;eRFID[66].bCapCorrectChecked;	eRFID[66].bCapCorrectCheckCameraOK;		eRFID[66].bCapCorrectCheckCameraChecked;		eRFID[66].bCapCorrectCapOn;eRFID[66].bCapCorrectNOK; eRFID[66].bFormPresent; eRFID[66].bBottlePresent; eRFID[66].bDosingTwoPhases; eRFID[66].nDispencerNr; eRFID[66].nDispencerNrSecondPhase; eRFID[66].lrDoseVolumeSV; eRFID[66].lrDoseVolumeCV; eRFID[66].lrDoseVolumeSVSecondPhase; eRFID[66].lrDoseVolumeCVSecondPhase; eRFID[66].bDosed;	eRFID[66].bDoseAborted; eRFID[66].bWeighed; eRFID[66].lrWeightSV; eRFID[66].lrWeightCV; eRFID[66].lrWeightMeasuredCV; eRFID[66].bWeightOK; eRFID[66].bCapPutted; eRFID[66].bCapChecked; eRFID[66].bCapOK; eRFID[66].bCapGripperScrewed; eRFID[66].bCapGripperScrewAborted; eRFID[66].bBottleTransferedToExit; eRFID[66].bBottleTransferedToLabeler; eRFID[66].lrWeightDif; eRFID[66].lrMinWeightCV;eRFID[66].lrMaxWeightCV;
eRFID[67].nCardNumber;eRFID[67].bCapCorrectChecked;	eRFID[67].bCapCorrectCheckCameraOK;		eRFID[67].bCapCorrectCheckCameraChecked;		eRFID[67].bCapCorrectCapOn;eRFID[67].bCapCorrectNOK; eRFID[67].bFormPresent; eRFID[67].bBottlePresent; eRFID[67].bDosingTwoPhases; eRFID[67].nDispencerNr; eRFID[67].nDispencerNrSecondPhase; eRFID[67].lrDoseVolumeSV; eRFID[67].lrDoseVolumeCV; eRFID[67].lrDoseVolumeSVSecondPhase; eRFID[67].lrDoseVolumeCVSecondPhase; eRFID[67].bDosed;	eRFID[67].bDoseAborted; eRFID[67].bWeighed; eRFID[67].lrWeightSV; eRFID[67].lrWeightCV; eRFID[67].lrWeightMeasuredCV; eRFID[67].bWeightOK; eRFID[67].bCapPutted; eRFID[67].bCapChecked; eRFID[67].bCapOK; eRFID[67].bCapGripperScrewed; eRFID[67].bCapGripperScrewAborted; eRFID[67].bBottleTransferedToExit; eRFID[67].bBottleTransferedToLabeler; eRFID[67].lrWeightDif; eRFID[67].lrMinWeightCV;eRFID[67].lrMaxWeightCV;
